(* CODESYS project Checkers.project

Project tree, tasks and I/O mapping:
  Device : PAC320-CXX2X-XX, Parker Hannifin, order no. PAC320-CXX2X-XX, version 3.5.9.10
    application Application
      libraries: Standard, * (System)
      task MainTask (externalevent, external event EVENT_ECM_DC, priority 0) calls EtherCAT_Master.EtherCAT_Task [EtherCAT_Master.EtherCAT_Task], Gameplay, TurnEnforcer, KingTextControl, TestPower, MakeMove, AxisPositionFeedback
      task VISU_TASK (cyclic, interval 100 ms, priority 31) calls VisuElems.Visu_Prg
      data type Piece
      data type BoardSpace
      program HMISequence [SFC]
      visualisation Loading_Screen
      visualisation Home_Screen
      program Gameplay [ST]
      function placePiece [ST]
      program ProgramFlow [SFC]
      visualisation Checkerboard
      function movePieceToStart [ST]
      program Init [ST]
      function pop [ST]
      function assignStartingPositions [ST]
      function checkForJumpRed1 [ST]
      function movePiece [ST]
      function pieceSelect [ST]
      function checkForJumpRed2 [ST]
      global variables GVL
      program TurnEnforcer [ST]
      program MakeMove [ST]
      program UpdateValidMoveArrays [ST]
      function checkForJumpRed3 [ST]
      function checkForJumpRed4 [ST]
      program ClearTakenPieces [ST]
      function checkForJumpBlack1 [ST]
      function checkForJumpBlack2 [ST]
      function checkForJumpBlack3 [ST]
      function checkForJumpBlack4 [ST]
      data type JumpProfile
      function clearJumpArr [ST]
      program KingTextControl [ST]
      program JumpPieces [ST]
      data type JumpDetail
      function push [ST]
      function clearGlobalStack [ST]
      function findSelectedPiece [ST]
      program MakeJump [ST]
      function findPieceAtGivenLocation [ST]
      function clearPieceJumpArray [ST]
      axis group XYZ: TRAFO.Kin_Gantry3, axes X, Y, Z
      SymbolConfiguration
      function block MovePieceMotion [CFC]
      program TestPower [CFC]
      program AxisPositionFeedback [CFC]
      function block timeDelay [CFC]
    SoftMotion General Axis Pool
    EtherCAT_Master : PAC320 EtherCAT Master, Parker Hannifin, order no. PAC320-XXXXX-XX, version 3.5.9.10
      PAC320_BusCoupler : PAC320 BusCoupler, Parker Hannifin, version Revision=16#00000001
          settings: StationAlias = 0; DC sync0 cycletime = 4000; DC sync1 cycletime = 4000
        PACIO_DI16_DO16 : DI16/DO16 1ms 0.5A (PACIO-450-03), Parker Hannifin, version Revision=16#00000001
            settings: StationAlias = 0; DC sync0 cycletime = 4000; DC sync1 cycletime = 4000
            unmapped channels: DigitalOutput0, DigitalOutput1, DigitalOutput2, DigitalOutput3, DigitalOutput4, DigitalOutput5, DigitalOutput6, DigitalOutput7, DigitalOutput8, DigitalOutput9, DigitalOutput10, DigitalOutput11, DigitalOutput12, DigitalOutput13, DigitalOutput14, DigitalOutput15, DigitalInput0, DigitalInput1, DigitalInput2, DigitalInput3, DigitalInput4, DigitalInput5, DigitalInput6, DigitalInput7, DigitalInput8, DigitalInput9, DigitalInput10, DigitalInput11, DigitalInput12, DigitalInput13, DigitalInput14, DigitalInput15
        PACIO_DI16_DO16_1 : DI16/DO16 1ms 0.5A LS (PACIO-450-13), Parker Hannifin, version Revision=16#00000001
            settings: DC sync0 cycletime = 4000; DC sync1 cycletime = 4000
            output GripperMove : BIT  // DigitalOutput0
            unmapped channels: DigitalOutput1, DigitalOutput2, DigitalOutput3, DigitalOutput4, DigitalOutput5, DigitalOutput6, DigitalOutput7, DigitalOutput8, DigitalOutput9, DigitalOutput10, DigitalOutput11, DigitalOutput12, DigitalOutput13, DigitalOutput14, DigitalOutput15, DigitalInput0, DigitalInput1, DigitalInput2, DigitalInput3, DigitalInput4, DigitalInput5, DigitalInput6, DigitalInput7, DigitalInput8, DigitalInput9, DigitalInput10, DigitalInput11, DigitalInput12, DigitalInput13, DigitalInput14, DigitalInput15
      PD_xxC_Standard_EtherCAT_drive : PD-xxC - Standard EtherCAT drive(CoE,EoE,FoE) V2.0, Parker Hannifin, version Revision=16#00000002
          settings: StationAlias = 0; DC sync0 cycletime = 4000
          unmapped channels: Controlword, Target Position, Touch Probe Function, Digital Ouputs, Statusword, Position Actual Value, Following Error Actual Value, Touch Probe Status, Touch Probe 1 Positive Edge Position Value, Digital Inputs
        X : SM_Drive_GenericDSP402, 3S - Smart Software Solutions GmbH, order no. 0, version 4.0.0.0
            settings: wDriveID = 0; dwRatioTechUnitsDenom = 3670016; iRatioTechUnitsNum = -125; fSWMaxVelocity = 100; ScalingIncs = 524288; ScalingMotorTurns2 = 7; ScalingUnits = 125; InvertDirection = TRUE; AdrOffset_8010 = 4; BitOffset_8010 = 0; BitLength_8010 = 16; Address_8010 = '%QW2'; Type_8010 = 'UINT'; AddressPointer_8010 = ADR(%QW2); AdrOffset_8020 = 8; BitOffset_8020 = 0; BitLength_8020 = 32; Address_8020 = '%QD2'; Type_8020 = 'DINT'; AddressPointer_8020 = ADR(%QD2); AdrOffset_8030 = 4294967295; BitOffset_8030 = 0; BitLength_8030 = 0; Address_8030 = ''; Type_8030 = ''; AddressPointer_8030 = 0; AdrOffset_8040 = 4294967295; BitOffset_8040 = 0; BitLength_8040 = 0; Address_8040 = ''; Type_8040 = ''; AddressPointer_8040 = 0; AdrOffset_8050 = 4294967295; BitOffset_8050 = 0; BitLength_8050 = 0; Address_8050 = ''; Type_8050 = ''; AddressPointer_8050 = 0; AdrOffset_8060 = 12; BitOffset_8060 = 0;
              BitLength_8060 = 16; Address_8060 = '%QW6'; Type_8060 = 'UINT'; AddressPointer_8060 = ADR(%QW6); AdrOffset_8070 = 4294967295; BitOffset_8070 = 0; BitLength_8070 = 0; Address_8070 = ''; Type_8070 = ''; AddressPointer_8070 = 0; AdrOffset_8080 = 4294967295; BitOffset_8080 = 0; BitLength_8080 = 0; Address_8080 = ''; Type_8080 = ''; AddressPointer_8080 = 0; AdrOffset_8090 = 16; BitOffset_8090 = 0; BitLength_8090 = 32; Address_8090 = '%QD4'; Type_8090 = 'UDINT'; AddressPointer_8090 = ADR(%QD4); AdrOffset_8510 = 4; BitOffset_8510 = 0; BitLength_8510 = 16; Address_8510 = '%IW2'; Type_8510 = 'UINT'; AddressPointer_8510 = ADR(%IW2); AdrOffset_8520 = 8; BitOffset_8520 = 0; BitLength_8520 = 32; Address_8520 = '%ID2'; Type_8520 = 'DINT'; AddressPointer_8520 = ADR(%ID2); AdrOffset_8530 = 4294967295; BitOffset_8530 = 0; BitLength_8530 = 0; Address_8530 = ''; Type_8530 = ''; AddressPointer_8530 = 0;
              AdrOffset_8540 = 4294967295; BitOffset_8540 = 0; BitLength_8540 = 0; Address_8540 = ''; Type_8540 = ''; AddressPointer_8540 = 0; AdrOffset_8550 = 4294967295; BitOffset_8550 = 0; BitLength_8550 = 0; Address_8550 = ''; Type_8550 = ''; AddressPointer_8550 = 0; AdrOffset_8560 = 24; BitOffset_8560 = 0; BitLength_8560 = 32; Address_8560 = '%ID6'; Type_8560 = 'UDINT'; AddressPointer_8560 = ADR(%ID6); AdrOffset_8570 = 16; BitOffset_8570 = 0; BitLength_8570 = 16; Address_8570 = '%IW8'; Type_8570 = 'UINT'; AddressPointer_8570 = ADR(%IW8); AdrOffset_8580 = 20; BitOffset_8580 = 0; BitLength_8580 = 32; Address_8580 = '%ID5'; Type_8580 = 'DINT'; AddressPointer_8580 = ADR(%ID5); AdrOffset_8590 = 4294967295; BitOffset_8590 = 0; BitLength_8590 = 0; Address_8590 = ''; Type_8590 = ''; AddressPointer_8590 = 0; AdrOffset_8600 = 4294967295; BitOffset_8600 = 0; BitLength_8600 = 0; Address_8600 = '';
              Type_8600 = ''; AddressPointer_8600 = 0; AdrOffset_8600 = 4294967295; BitOffset_8600 = 0; BitLength_8600 = 0; Address_8610 = ''; Type_8610 = ''; AddressPointer_8610 = 0; AdrOffset_8620 = 12; BitOffset_8620 = 0; BitLength_8620 = 32; Address_8620 = '%ID3'; Type_8620 = 'DINT'; AddressPointer_8620 = ADR(%ID3)
      PD_xxC_Standard_EtherCAT_drive_1 : PD-xxC - Standard EtherCAT drive(CoE,EoE,FoE) V2.0, Parker Hannifin, version Revision=16#00000002
          settings: StationAlias = 0; DC sync0 cycletime = 4000
          unmapped channels: Controlword, Target Position, Touch Probe Function, Digital Ouputs, Statusword, Position Actual Value, Following Error Actual Value, Touch Probe Status, Touch Probe 1 Positive Edge Position Value, Digital Inputs
        Y : SM_Drive_GenericDSP402, 3S - Smart Software Solutions GmbH, order no. 0, version 4.0.0.0
            settings: dwRatioTechUnitsDenom = 65536; iRatioTechUnitsNum = 3; fSWMaxVelocity = 100; ScalingIncs = 262144; ScalingMotorTurns2 = 5; ScalingUnits = 60; AdrOffset_8010 = 20; BitOffset_8010 = 0; BitLength_8010 = 16; Address_8010 = '%QW10'; Type_8010 = 'UINT'; AddressPointer_8010 = ADR(%QW10); AdrOffset_8020 = 24; BitOffset_8020 = 0; BitLength_8020 = 32; Address_8020 = '%QD6'; Type_8020 = 'DINT'; AddressPointer_8020 = ADR(%QD6); AdrOffset_8030 = 4294967295; BitOffset_8030 = 0; BitLength_8030 = 0; Address_8030 = ''; Type_8030 = ''; AddressPointer_8030 = 0; AdrOffset_8040 = 4294967295; BitOffset_8040 = 0; BitLength_8040 = 0; Address_8040 = ''; Type_8040 = ''; AddressPointer_8040 = 0; AdrOffset_8050 = 4294967295; BitOffset_8050 = 0; BitLength_8050 = 0; Address_8050 = ''; Type_8050 = ''; AddressPointer_8050 = 0; AdrOffset_8060 = 28; BitOffset_8060 = 0; BitLength_8060 = 16; Address_8060 = '%QW14';
              Type_8060 = 'UINT'; AddressPointer_8060 = ADR(%QW14); AdrOffset_8070 = 4294967295; BitOffset_8070 = 0; BitLength_8070 = 0; Address_8070 = ''; Type_8070 = ''; AddressPointer_8070 = 0; AdrOffset_8080 = 4294967295; BitOffset_8080 = 0; BitLength_8080 = 0; Address_8080 = ''; Type_8080 = ''; AddressPointer_8080 = 0; AdrOffset_8090 = 32; BitOffset_8090 = 0; BitLength_8090 = 32; Address_8090 = '%QD8'; Type_8090 = 'UDINT'; AddressPointer_8090 = ADR(%QD8); AdrOffset_8510 = 28; BitOffset_8510 = 0; BitLength_8510 = 16; Address_8510 = '%IW14'; Type_8510 = 'UINT'; AddressPointer_8510 = ADR(%IW14); AdrOffset_8520 = 32; BitOffset_8520 = 0; BitLength_8520 = 32; Address_8520 = '%ID8'; Type_8520 = 'DINT'; AddressPointer_8520 = ADR(%ID8); AdrOffset_8530 = 4294967295; BitOffset_8530 = 0; BitLength_8530 = 0; Address_8530 = ''; Type_8530 = ''; AddressPointer_8530 = 0; AdrOffset_8540 = 4294967295; BitOffset_8540 = 0;
              BitLength_8540 = 0; Address_8540 = ''; Type_8540 = ''; AddressPointer_8540 = 0; AdrOffset_8550 = 4294967295; BitOffset_8550 = 0; BitLength_8550 = 0; Address_8550 = ''; Type_8550 = ''; AddressPointer_8550 = 0; AdrOffset_8560 = 48; BitOffset_8560 = 0; BitLength_8560 = 32; Address_8560 = '%ID12'; Type_8560 = 'UDINT'; AddressPointer_8560 = ADR(%ID12); AdrOffset_8570 = 40; BitOffset_8570 = 0; BitLength_8570 = 16; Address_8570 = '%IW20'; Type_8570 = 'UINT'; AddressPointer_8570 = ADR(%IW20); AdrOffset_8580 = 44; BitOffset_8580 = 0; BitLength_8580 = 32; Address_8580 = '%ID11'; Type_8580 = 'DINT'; AddressPointer_8580 = ADR(%ID11); AdrOffset_8590 = 4294967295; BitOffset_8590 = 0; BitLength_8590 = 0; Address_8590 = ''; Type_8590 = ''; AddressPointer_8590 = 0; AdrOffset_8600 = 4294967295; BitOffset_8600 = 0; BitLength_8600 = 0; Address_8600 = ''; Type_8600 = ''; AddressPointer_8600 = 0;
              AdrOffset_8600 = 4294967295; BitOffset_8600 = 0; BitLength_8600 = 0; Address_8610 = ''; Type_8610 = ''; AddressPointer_8610 = 0; AdrOffset_8620 = 36; BitOffset_8620 = 0; BitLength_8620 = 32; Address_8620 = '%ID9'; Type_8620 = 'DINT'; AddressPointer_8620 = ADR(%ID9)
      PD_xxC_Standard_EtherCAT_drive_2 : PD-xxC - Standard EtherCAT drive(CoE,EoE,FoE) V2.0, Parker Hannifin, version Revision=16#00000002
          settings: StationAlias = 0; DC sync0 cycletime = 4000
          unmapped channels: Controlword, Target Position, Touch Probe Function, Digital Ouputs, Statusword, Position Actual Value, Following Error Actual Value, Touch Probe Status, Touch Probe 1 Positive Edge Position Value, Digital Inputs
        Z : SM_Drive_GenericDSP402, 3S - Smart Software Solutions GmbH, order no. 0, version 4.0.0.0
            settings: wDriveID = 2; dwRatioTechUnitsDenom = 262144; iRatioTechUnitsNum = 5; fSWMaxVelocity = 100; fSWMaxAcceleration = 500; fSWMaxDeceleration = 500; fSWMaxJerk = 5000; ScalingIncs = 262144; ScalingUnits = 5; AdrOffset_8010 = 36; BitOffset_8010 = 0; BitLength_8010 = 16; Address_8010 = '%QW18'; Type_8010 = 'UINT'; AddressPointer_8010 = ADR(%QW18); AdrOffset_8020 = 40; BitOffset_8020 = 0; BitLength_8020 = 32; Address_8020 = '%QD10'; Type_8020 = 'DINT'; AddressPointer_8020 = ADR(%QD10); AdrOffset_8030 = 4294967295; BitOffset_8030 = 0; BitLength_8030 = 0; Address_8030 = ''; Type_8030 = ''; AddressPointer_8030 = 0; AdrOffset_8040 = 4294967295; BitOffset_8040 = 0; BitLength_8040 = 0; Address_8040 = ''; Type_8040 = ''; AddressPointer_8040 = 0; AdrOffset_8050 = 4294967295; BitOffset_8050 = 0; BitLength_8050 = 0; Address_8050 = ''; Type_8050 = ''; AddressPointer_8050 = 0; AdrOffset_8060 = 44;
              BitOffset_8060 = 0; BitLength_8060 = 16; Address_8060 = '%QW22'; Type_8060 = 'UINT'; AddressPointer_8060 = ADR(%QW22); AdrOffset_8070 = 4294967295; BitOffset_8070 = 0; BitLength_8070 = 0; Address_8070 = ''; Type_8070 = ''; AddressPointer_8070 = 0; AdrOffset_8080 = 4294967295; BitOffset_8080 = 0; BitLength_8080 = 0; Address_8080 = ''; Type_8080 = ''; AddressPointer_8080 = 0; AdrOffset_8090 = 48; BitOffset_8090 = 0; BitLength_8090 = 32; Address_8090 = '%QD12'; Type_8090 = 'UDINT'; AddressPointer_8090 = ADR(%QD12); AdrOffset_8510 = 52; BitOffset_8510 = 0; BitLength_8510 = 16; Address_8510 = '%IW26'; Type_8510 = 'UINT'; AddressPointer_8510 = ADR(%IW26); AdrOffset_8520 = 56; BitOffset_8520 = 0; BitLength_8520 = 32; Address_8520 = '%ID14'; Type_8520 = 'DINT'; AddressPointer_8520 = ADR(%ID14); AdrOffset_8530 = 4294967295; BitOffset_8530 = 0; BitLength_8530 = 0; Address_8530 = ''; Type_8530 = '';
              AddressPointer_8530 = 0; AdrOffset_8540 = 4294967295; BitOffset_8540 = 0; BitLength_8540 = 0; Address_8540 = ''; Type_8540 = ''; AddressPointer_8540 = 0; AdrOffset_8550 = 4294967295; BitOffset_8550 = 0; BitLength_8550 = 0; Address_8550 = ''; Type_8550 = ''; AddressPointer_8550 = 0; AdrOffset_8560 = 72; BitOffset_8560 = 0; BitLength_8560 = 32; Address_8560 = '%ID18'; Type_8560 = 'UDINT'; AddressPointer_8560 = ADR(%ID18); AdrOffset_8570 = 64; BitOffset_8570 = 0; BitLength_8570 = 16; Address_8570 = '%IW32'; Type_8570 = 'UINT'; AddressPointer_8570 = ADR(%IW32); AdrOffset_8580 = 68; BitOffset_8580 = 0; BitLength_8580 = 32; Address_8580 = '%ID17'; Type_8580 = 'DINT'; AddressPointer_8580 = ADR(%ID17); AdrOffset_8590 = 4294967295; BitOffset_8590 = 0; BitLength_8590 = 0; Address_8590 = ''; Type_8590 = ''; AddressPointer_8590 = 0; AdrOffset_8600 = 4294967295; BitOffset_8600 = 0; BitLength_8600 = 0;
              Address_8600 = ''; Type_8600 = ''; AddressPointer_8600 = 0; AdrOffset_8600 = 4294967295; BitOffset_8600 = 0; BitLength_8600 = 0; Address_8610 = ''; Type_8610 = ''; AddressPointer_8610 = 0; AdrOffset_8620 = 60; BitOffset_8620 = 0; BitLength_8620 = 32; Address_8620 = '%ID15'; Type_8620 = 'DINT'; AddressPointer_8620 = ADR(%ID15)
  text list GlobalTextList
*)

// Device/Application/Piece
TYPE Piece :
STRUCT
	isBlack : BOOL := FALSE; // False indicates that a piece is red; true indicates black
	isTaken : BOOL := FALSE; // False indicates that a piece is still in play
	isKing : BOOL := FALSE; // True indicates that a piece is a king
	isSelected : BOOL := FALSE;
	oldLocation : ARRAY [0..1] OF INT := [0,0];
	currentLocation : ARRAY [0..1] OF INT := [0,0]; // -1, -1 indicated that the piece has been taken
	translatedLocation : ARRAY [0..1] OF INT; // translated movement in terms of HMI coordinates
	startingLocation : ARRAY [0..1] OF INT;
	validMoveArr : ARRAY [0..7,0..7] OF BOOL; // 2D array represents the board, true indicates that a piece can move to that space 
	
	jumpArr : ARRAY [0..20,0..3] OF JumpDetail;
	
	startStack : INT;
	jumpedPieceIndex : INT;
	kingText : WSTRING := "";
END_STRUCT
END_TYPE

// Device/Application/BoardSpace
TYPE BoardSpace :
STRUCT
	isBlack : BOOL := FALSE;
	isRed : BOOL := FALSE;
	isEmpty : BOOL := TRUE;
	chosenForMove : BOOL := FALSE;
	
	xLoc : INT;
END_STRUCT
END_TYPE

// Device/Application/JumpProfile
TYPE JumpProfile :
STRUCT
	jumpRef : INT;
	lastJumpRef : INT := -1;
	xMoveLocation : INT;
	yMoveLocation : INT;
	xJumpedLocation : INT;
	yJumpedLocation : INT;
	numPiecesToJump : INT;
	jumpedPieceColor : INT;
	jumpedPieceIndex : INT;
	jumpingPieceX : INT;
	jumpingPieceY : INT;
END_STRUCT
END_TYPE

// Device/Application/JumpDetail
TYPE JumpDetail :
STRUCT
	
	xMoveLocation : INT := -1;
	yMoveLocation : INT := -1;
	jumpedColor : INT := -1;
	jumpedIndex : INT := -1;
	
	
END_STRUCT
END_TYPE

// Device/Application/GVL
{attribute 'qualified_only'}
VAR_GLOBAL
	selectedPieceValidMoveArr : ARRAY [0..7,0..7] OF BOOL;
	noValidMoveArr : ARRAY [0..7,0..7] OF BOOL;
	selectedPieceValidJumpArr : ARRAY [0..7,0..7] OF BOOL;
	board : ARRAY [0..7,0..7] OF BoardSpace; // represents every space on the board
	pieces : ARRAY [0..1,0..11] OF Piece; // 1,x is any black piece, 0,x is any red piece
	redsTurn : BOOL := TRUE;
	
	jumpMoveArr : ARRAY[0..100] OF JumpProfile;
	currentJumpRef : INT := 0;
	
	xMoveSpace : INT := -1;
	yMoveSpace : INT := -1;
	
	boardIsSetup : BOOL;
	
	takenList : ARRAY [0..20,0..1] OF INT;
	takenListLength : INT;
	emptyTakenList : ARRAY [0..20,0..1] OF INT;
	
	jumpStack : ARRAY[0..3] OF JumpDetail;
	currentStackIndex : INT;
	currentJumpProfileNum : INT;
	
	emptyJumpArr : ARRAY [0..20,0..3] OF JumpDetail;
	
	redStack0Offset : ARRAY [0..1] OF INT := [0,100]; // coordinate offset of red stacks in HMI (at beginning of game)
	redStack1Offset : ARRAY [0..1] OF INT := [100,100]; // coordinate offset of red stacks in HMI (at beginning of game)
	redStack2Offset : ARRAY [0..1] OF INT := [200, 100]; // coordinate offset of red stacks in HMI (at beginning of game)
	
	blackStack0Offset : ARRAY [0..1] OF INT := [350,-450];
	blackStack1Offset : ARRAY [0..1] OF INT := [250,-450];
	blackStack2Offset : ARRAY [0..1] OF INT := [150,-450];
	
	redPiecesTaken : INT := 0;
	blackPiecesTaken : INT := 0;
	
	test : BOOL := FALSE;
	
END_VAR

// Device/Application/Gameplay
PROGRAM Gameplay
VAR
	//selectedPieceValidMoveArr : ARRAY [0..7,0..7] OF BOOL;
	//noValidMoveArr : ARRAY [0..7,0..7] OF BOOL;
	//board : ARRAY [0..7,0..7] OF BoardSpace; // represents every space on the board
	//pieces : ARRAY [0..1,0..11] OF Piece; // 0,x is any black piece, 1,x is any red piece
	startingPositionsRed : ARRAY [0..1,0..11] OF INT;
	startingPositionsBlack : ARRAY [0..1,0..11] OF INT;
	redIsAssigned : BOOL := FALSE;
	blackIsAssigned : BOOL := FALSE;
	
	// ****************VARIABLES FOR BOARD SETUP*******************
	numStacks : INT := 3;
	numPiecesInStack : INT := 5;
	numPieces : INT := 12;
	currentStack : INT := 0; // stack that gripper is currently drawing from
	currentPiece : INT := 0; // piece number that gripper has set up
	currentStackPos : INT := 0;	// stack position flows 0-4 from top to bottom
	currentSpace : ARRAY [0..1] OF INT;
	piecePosition : ARRAY[0..1] OF INT;
	
	done : BOOL;
	i : INT := 0;
	j : INT := 0;
	boardCleared : BOOL := FALSE;
	y: INT;
	pieceNum: INT;
	x: INT;
	temp : INT;
	commenceSetup : BOOL := FALSE; // Variable toggled by pushing the set up board button
	xPos: INT;
	yPos: INT;
	found : BOOL := FALSE;
END_VAR

IF(commenceSetup) THEN
	IF(NOT GVL.boardIsSetup) THEN
	

		// Assigns starting positions for red and black GVL.pieces
	IF(NOT redIsAssigned) THEN
		startingPositionsRed := assignStartingPositions(startingPositionsRed, TRUE);
		redIsAssigned := TRUE;
	END_IF
	IF(NOT blackIsAssigned) THEN
		startingPositionsBlack := assignStartingPositions(startingPositionsBlack, FALSE);
		blackIsAssigned := TRUE;
	END_IF


	// initializes values for red GVL.pieces
	FOR i := 0 TO (numPieces - 1) DO
		GVL.pieces[0,i].isBlack := FALSE;
		GVL.pieces[0,i].isKing := FALSE;
		GVL.pieces[0,i].isTaken := FALSE;
		GVL.pieces[0,i].currentLocation[0] := startingPositionsRed[0,i]; 
		GVL.pieces[0,i].currentLocation[1] := startingPositionsRed[1,i];
		GVL.pieces[0,i].jumpedPieceIndex := i;
		IF(i < numPiecesInStack) THEN
			GVL.pieces[0,i].startStack := 0;
		ELSIF(i < (numPiecesInStack * 2) AND i >= numPiecesInStack) THEN
			GVL.pieces[0,i].startStack := 1;
		ELSE
			GVL.pieces[0,i].startStack := 2;
		END_IF
		GVL.pieces[0,i] := movePieceToStart(GVL.pieces[0,i]);
		GVL.board[GVL.pieces[0,i].currentLocation[0], GVL.pieces[0,i].currentLocation[1]].isRed := TRUE;
		GVL.board[GVL.pieces[0,i].currentLocation[0], GVL.pieces[0,i].currentLocation[1]].isBlack := FALSE;
		GVL.board[GVL.pieces[0,i].currentLocation[0], GVL.pieces[0,i].currentLocation[1]].isEmpty := FALSE;
	END_FOR


	// initializes values for black GVL.pieces
	FOR i := 0 TO (numPieces - 1) DO
		GVL.pieces[1,i].isBlack := TRUE;
		GVL.pieces[1,i].isKing := FALSE;
		GVL.pieces[1,i].isTaken := FALSE;
		GVL.pieces[1,i].currentLocation[0] := startingPositionsBlack[0,i];
		GVL.pieces[1,i].currentLocation[1] := startingPositionsBlack[1,i];
		IF(i < numPiecesInStack) THEN
			GVL.pieces[1,i].startStack := 0;
		ELSIF(i < (numPiecesInStack * 2) AND i >= numPiecesInStack) THEN
			GVL.pieces[1,i].startStack := 1;
		ELSE
			GVL.pieces[1,i].startStack := 2;
		END_IF
		GVL.pieces[1,i] := movePieceToStart(GVL.pieces[1,i]);
		GVL.board[GVL.pieces[1,i].currentLocation[0], GVL.pieces[1,i].currentLocation[1]].isRed := FALSE;
		GVL.board[GVL.pieces[1,i].currentLocation[0], GVL.pieces[1,i].currentLocation[1]].isBlack := TRUE;
		GVL.board[GVL.pieces[1,i].currentLocation[0], GVL.pieces[1,i].currentLocation[1]].isEmpty := FALSE;
	END_FOR

	GVL.boardIsSetup := TRUE;
END_IF

// Setup valid moves for red
FOR i:= 0 TO numPieces - 1 DO
	x:= GVL.pieces[0,i].currentLocation[0];
	y := GVL.pieces[0,i].currentLocation[1];
	
	// Checks for move up and right
	IF(x+1 < 8 AND y+1 < 8 AND GVL.board[x+1,y+1].isEmpty) THEN
		GVL.pieces[0,i].validMoveArr[x+1,y+1] := TRUE;
	END_IF

	// Checks for move up and left
	IF(x-1 >= 0 AND y+1 < 8 AND GVL.board[x-1,y+1].isEmpty) THEN
		GVL.pieces[0,i].validMoveArr[x-1,y+1] := TRUE;
	END_IF
	
	IF(x+1 < 8 AND y+1 < 8 AND NOT GVL.board[x+1,y+1].isEmpty AND GVL.board[x+1,y+1].isBlack) THEN
		
		//possible jump
	END_IF
	
END_FOR

// Setup valid moves for black
FOR i:= 0 TO numPieces - 1 DO
	x:= GVL.pieces[1,i].currentLocation[0];
	y := GVL.pieces[1,i].currentLocation[1];
	
	// Checks for move up and right
	IF(x+1 < 8 AND y+1 < 8 AND GVL.board[x+1,y-1].isEmpty) THEN
		GVL.pieces[1,i].validMoveArr[x+1,y-1] := TRUE;
	END_IF

	// Checks for move up and left
	IF(x-1 >= 0 AND y+1 < 8 AND GVL.board[x-1,y-1].isEmpty) THEN
		GVL.pieces[1,i].validMoveArr[x-1,y-1] := TRUE;
	END_IF
	
	(*
	IF(x+1 < 8 AND y+1 < 8 AND NOT GVL.board[x+1,y+1].isEmpty AND GVL.board[x+1,y+1].isBlack) THEN
		
		//possible jump
	END_IF
	*)
	
END_FOR



END_IF

END_PROGRAM

// Device/Application/assignStartingPositions
FUNCTION assignStartingPositions : ARRAY [0..1,0..11] OF INT;
VAR_INPUT
	startingPos : ARRAY [0..1,0..11] OF INT;
	isRed : BOOL;
END_VAR
VAR
	numPieces : INT := 12;
	
	i: INT;
	y: INT;
	x: INT;
	temp: INT;
END_VAR

IF(isRed) THEN
	FOR i := 0 TO (numPieces - 1) DO 	
		y := i / 4;
		x := ((2 * i) MOD 8) + (y MOD 2);
		startingPos[0,i] := x;
		startingPos[1,i] := y;
	END_FOR
ELSE
	FOR i := 0 TO (numPieces - 1) DO 
		temp := i / 4;
		x := ((2 * i) MOD 8) + (temp MOD 2);
		y := temp + 5;
		x := x + 1;
		IF(x >= 8) THEN
			x := x MOD 8;
		END_IF
		startingPos[0,i] := x;
		startingPos[1,i] := y;	
	END_FOR
END_IF

assignStartingPositions := startingPos;
RETURN;

END_FUNCTION

// Device/Application/movePieceToStart
FUNCTION movePieceToStart : Piece
VAR_INPUT
	currentPiece : Piece;
END_VAR
VAR
	
	spaceTranslation : ARRAY [0..1] OF INT; // small numbers (0-7) that indicate how many spaces a piece needs to be moved
	sizeOfMoveX : INT := 50;
	sizeOfMoveY : INT := -50;
END_VAR

movePieceToStart := currentPiece;
IF(NOT movePieceToStart.isBlack) THEN
	// Moves pieces from their stack to the origin (board sqaure 0,0 or bottom left corner)
	IF(currentPiece.startStack = 0) THEN
		movePieceToStart.translatedLocation[0] := currentPiece.translatedLocation[0] - GVL.redStack0Offset[0];
		movePieceToStart.translatedLocation[1] := currentPiece.translatedLocation[1] - GVL.redStack0Offset[1];
		
	ELSIF(currentPiece.startStack = 1) THEN
		movePieceToStart.translatedLocation[0] := currentPiece.translatedLocation[0] - GVL.redStack1Offset[0];
		movePieceToStart.translatedLocation[1] := currentPiece.translatedLocation[1] - GVL.redStack1Offset[1];
	ELSE
		movePieceToStart.translatedLocation[0] := currentPiece.translatedLocation[0] - GVL.redStack2Offset[0];
		movePieceToStart.translatedLocation[1] := currentPiece.translatedLocation[1] - GVL.redStack2Offset[1];
	END_IF
ELSE
	IF(currentPiece.startStack = 0) THEN
		movePieceToStart.translatedLocation[0] := currentPiece.translatedLocation[0] - GVL.blackStack0Offset[0];
		movePieceToStart.translatedLocation[1] := currentPiece.translatedLocation[1] - GVL.blackStack0Offset[1];
	ELSIF(currentPiece.startStack = 1) THEN
		movePieceToStart.translatedLocation[0] := currentPiece.translatedLocation[0] - GVL.blackStack1Offset[0];
		movePieceToStart.translatedLocation[1] := currentPiece.translatedLocation[1] - GVL.blackStack1Offset[1];
	ELSE
		movePieceToStart.translatedLocation[0] := currentPiece.translatedLocation[0] - GVL.blackStack2Offset[0];
		movePieceToStart.translatedLocation[1] := currentPiece.translatedLocation[1] - GVL.blackStack2Offset[1];
	END_IF			

END_IF

movePieceToStart.startingLocation := movePieceToStart.translatedLocation;

spaceTranslation[0] := movePieceToStart.currentLocation[0] - movePieceToStart.oldLocation[0];
spaceTranslation[1] := movePieceToStart.currentLocation[1] - movePieceToStart.oldLocation[1];

movePieceToStart.translatedLocation[0] := movePieceToStart.translatedLocation[0] + (spaceTranslation[0] * sizeOfMoveX);
movePieceToStart.translatedLocation[1] := movePieceToStart.translatedLocation[1] + (spaceTranslation[1] * sizeOfMoveY);

// set oldLocation to currentLocation
movePieceToStart.oldLocation[0] := movePieceToStart.currentLocation[0];
movePieceToStart.oldLocation[1] := movePieceToStart.currentLocation[1];


RETURN;

END_FUNCTION

// Device/Application/TurnEnforcer
PROGRAM TurnEnforcer
VAR
	i : INT;
	wrongColorSelected : BOOL;
END_VAR

// Stops user from selecting a piece that is taken
FOR i := 0 TO 11 DO
	IF(GVL.pieces[1,i].isTaken)THEN 
		GVL.pieces[1,i].isSelected := FALSE;
	ELSIF(GVL.pieces[0,i].isTaken) THEN
		GVL.pieces[0,i].isSelected := FALSE;
	END_IF
END_FOR

// Stops user from picking the wrong color
wrongColorSelected := FALSE;

IF(GVL.redsTurn) THEN
	FOR i := 0 TO 11 DO
		IF(GVL.pieces[1,i].isSelected)THEN 
			 GVL.pieces[1,i].isSelected := FALSE;
			 wrongColorSelected := TRUE;
		END_IF
	END_FOR
ELSE
	FOR i := 0 TO 11 DO
		IF(GVL.pieces[0,i].isSelected)THEN 
			 GVL.pieces[0,i].isSelected := FALSE;
			 wrongColorSelected := TRUE;
		END_IF				
	END_FOR
END_IF

IF(wrongColorSelected) THEN
	GVL.selectedPieceValidMoveArr := GVL.noValidMoveArr;
END_IF

END_PROGRAM

// Device/Application/KingTextControl
PROGRAM KingTextControl
VAR
	i : INT;
END_VAR

FOR i := 0 TO 11 DO
	IF(GVL.pieces[0,i].isKing) THEN
		GVL.pieces[0,i].kingText := "K";
	END_IF
	IF(GVL.pieces[1,i].isKing) THEN
		GVL.pieces[1,i].kingText := "K";
	END_IF
END_FOR

END_PROGRAM

// Device/Application/TestPower
PROGRAM TestPower
VAR
	xPower: MC_Power;
	yPower: MC_Power;
	zPower: MC_Power;
	EnableAxes: MC_GroupEnable;
	Enable: BOOL;
END_VAR

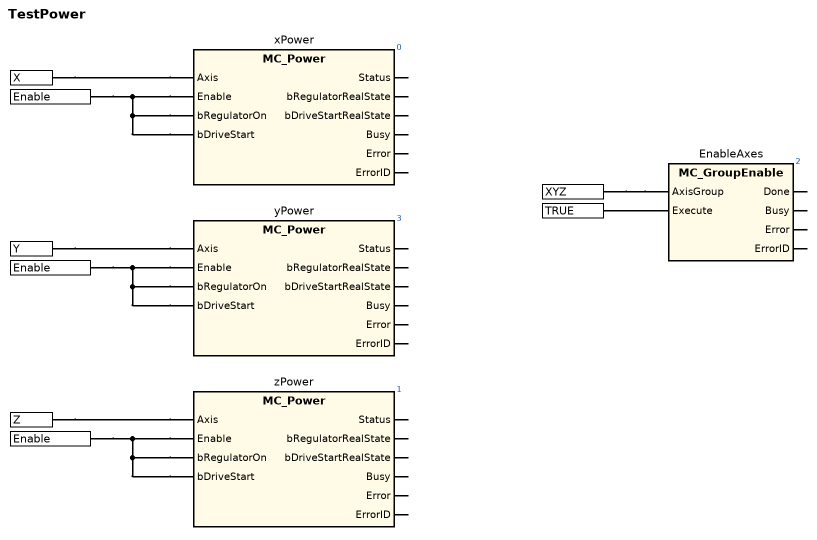
xPower(Axis := X, Enable := Enable, bRegulatorOn := Enable, bDriveStart := Enable); // MC_Power
zPower(Axis := Z, Enable := Enable, bRegulatorOn := Enable, bDriveStart := Enable); // MC_Power
EnableAxes(AxisGroup := XYZ, Execute := TRUE); // MC_GroupEnable
yPower(Axis := Y, Enable := Enable, bRegulatorOn := Enable, bDriveStart := Enable); // MC_Power

END_PROGRAM

// Device/Application/MakeMove
PROGRAM MakeMove
// moveSpace variables are only changed when a square is pushed in the HMI
VAR
	i : INT;
	counter : INT;
	xCurrentSpace : INT;
	yCurrentSpace : INT;
	currentPiece : Piece;
	selected : BOOL;
	redOrBlack : INT;
	jumpedPieceIndex : INT;
	
	spaceTranslation : ARRAY [0..1] OF INT; // small numbers (0-7) that indicate how many spaces a piece needs to be moved
	sizeOfMoveX : INT := 50;
	sizeOfMoveY : INT := -50;
	
	caseState : INT := 000;
	moveTest : MovePieceMotion;
	
	xOffset : LREAL := 100.455;
	yOffset : LREAL := -25.654;
	zUp : LREAL := 15;
	zDown: LREAL := 49;
	
	xStack : LREAL := 111;
	yStack : LREAL := -73;
	pieceOffset : LREAL := 6.36; 
	
	selectedPiece : ARRAY [0..1] OF INT;
	
	xPiece: INT;
	yPiece: INT;
	
	wait : timeDelay;
	
	jumpCounter : INT;

END_VAR

CASE caseState OF

// Will run in this case as long as a move space isn't selected
000:
	IF(GVL.xMoveSpace <> -1 AND GVL.yMoveSpace <> -1) THEN
		//GripperMove := FALSE;
		caseState := 001;
	END_IF
	
// If the move is valid, execution of the move begins by positioning
// the gripper over the piece that is to be moved
// If the move is invalid, case statement jumps back to case 000
001: 
	selectedPiece := findSelectedPiece();
	IF(GVL.selectedPieceValidMoveArr[GVL.xMoveSpace, GVL.yMoveSpace]) THEN
		xPiece := GVL.pieces[selectedPiece[0],selectedPiece[1]].currentLocation[0];
		yPiece := GVL.pieces[selectedPiece[0],selectedPiece[1]].currentLocation[1];
	
		moveTest.xPos := xOffset + (xPiece * 20);
		moveTest.yPos := yOffset + (yPiece * 20);
		moveTest.zPos := zUp;
	
		caseState := 002;
	ELSE
		// Deselects all pieces
		FOR i:=0 TO 11 DO
			GVL.pieces[0,i].isSelected := FALSE;
			GVL.pieces[1,i].isSelected := FALSE;			
		END_FOR
		GVL.xMoveSpace := -1;
		GVL.yMoveSpace := -1;
		
		caseState := 000;
	END_IF

// Move is executed	
002:
	moveTest.ExecuteMove := TRUE;
	caseState := 003;

// Once the gripper is in position above the piece to be moved
// execute move is set to false
003:
	IF(moveTest.MoveDone) THEN
		caseState := 004;
		moveTest.ExecuteMove := FALSE;
	END_IF

// Sets gripper to down position over the current piece
004:
	moveTest.zPos := zDown;
	caseState := 005;

005:
	moveTest.ExecuteMove := TRUE;
	caseState := 006;

// THIS IS WHERE THE PIECE WILL BE PICKED UP	
006:
	IF(moveTest.MoveDone)THEN
		caseState := 007;
		moveTest.ExecuteMove := FALSE;
		GripperMove := TRUE;
		wait.startTimer := TRUE;
	END_IF

007:
	IF(wait.done) THEN
		wait.startTimer := FALSE;
		moveTest.zPos := zUp;
		caseState := 008;
	END_IF
	
008: 
	moveTest.ExecuteMove := TRUE;
	caseState := 009;

009:
	IF(moveTest.MoveDone)THEN
		caseState := 010;
		moveTest.ExecuteMove := FALSE;
	END_IF
	
	
010:
	IF(GVL.xMoveSpace >= 0 AND GVL.yMoveSpace >= 0) THEN
		selected := FALSE;
		i := 0;
		// Figure out which piece is selected
		WHILE(i < 12 AND NOT selected) DO
		
			IF(GVL.pieces[0,i].isSelected) THEN
				xCurrentSpace := GVL.pieces[0,i].currentLocation[0];
				yCurrentSpace := GVL.pieces[0,i].currentLocation[1];
				currentPiece := GVL.pieces[0,i];
				redOrBlack := 0;
				jumpedPieceIndex := i;
				selected := TRUE;
			END_IF
			IF(GVL.pieces[1,i].isSelected) THEN
				xCurrentSpace := GVL.pieces[1,i].currentLocation[0];
				yCurrentSpace := GVL.pieces[1,i].currentLocation[1];
				currentPiece := GVL.pieces[1,i];
				redOrBlack := 1;
				jumpedPieceIndex := i;
				selected := TRUE;
			END_IF
			i := i + 1;
	
		END_WHILE
	
		// Determine if the move is legal
		IF(GVL.selectedPieceValidMoveArr[GVL.xMoveSpace, GVL.yMoveSpace])THEN 
			// Perform the move
			currentPiece.translatedLocation[0] := currentPiece.startingLocation[0] + (GVL.xMoveSpace * sizeOfMoveX);
			currentPiece.translatedLocation[1] := currentPiece.startingLocation[1] + (GVL.yMoveSpace * sizeOfMoveY);;
		
		
			moveTest.xPos := xOffset + (GVL.xMoveSpace * 20);
			moveTest.yPos := yOffset + (GVL.yMoveSpace * 20);
			moveTest.zPos := zUp;

			caseState := 020;
		
		
			// sets pieces current location as the old location, as it is about to move
			currentPiece.oldLocation[0] := currentPiece.currentLocation[0];
			currentPiece.oldLocation[1] := currentPiece.currentLocation[1];
	
			// updates the current location after the move has been completed
			currentPiece.currentLocation[0] := GVL.xMoveSpace;
			currentPiece.currentLocation[1] := GVL.yMoveSpace;
		
			// Piece is red and has achieved king status
			IF(currentPiece.currentLocation[1] = 7 AND NOT currentPiece.isBlack) THEN
				currentPiece.isKing := TRUE;
			// Piece is black and has achieved king status
			ELSIF(currentPiece.currentLocation[1] = 0 AND currentPiece.isBlack) THEN
				currentPiece.isKing := TRUE;
			END_IF
			
		
			// updates board space player just moved from
			GVL.board[currentPiece.oldLocation[0], currentPiece.oldLocation[1]].isEmpty := TRUE;
			GVL.board[currentPiece.oldLocation[0], currentPiece.oldLocation[1]].isBlack := FALSE;
			GVL.board[currentPiece.oldLocation[0], currentPiece.oldLocation[1]].isRed := FALSE;
		
			// updates board space that the player just moved to
			GVL.board[currentPiece.currentLocation[0], currentPiece.currentLocation[1]].isEmpty := FALSE;
			IF(currentPiece.isBlack)THEN
				GVL.board[currentPiece.currentLocation[0], currentPiece.currentLocation[1]].isBlack := TRUE;
				GVL.board[currentPiece.currentLocation[0], currentPiece.currentLocation[1]].isRed := FALSE;
			ELSE
				GVL.board[currentPiece.currentLocation[0], currentPiece.currentLocation[1]].isBlack := FALSE;
				GVL.board[currentPiece.currentLocation[0], currentPiece.currentLocation[1]].isRed := TRUE;
			END_IF
		
			GVL.pieces[redOrBlack, jumpedPieceIndex] := currentPiece;
		
		
		
			// Make it the other persons turn
			IF(GVL.redsTurn) THEN
				GVL.redsTurn := FALSE;
			ELSE
				GVL.redsTurn := TRUE;	
			END_IF
		
		
			MakeJump();
			UpdateValidMoveArrays();
		
			// Deselects all pieces
			GVL.selectedPieceValidMoveArr := GVL.noValidMoveArr;
			FOR i:=0 TO 11 DO
				GVL.pieces[0,i].isSelected := FALSE;
				GVL.pieces[1,i].isSelected := FALSE;			
			END_FOR
		
			IF(currentPiece.oldLocation[0] + 1 = currentPiece.currentLocation[0] OR
				currentPiece.oldLocation[1] + 1 = currentPiece.currentLocation[1] OR
				currentPiece.oldLocation[0] - 1 = currentPiece.currentLocation[0] OR
				currentPiece.oldLocation[1] - 1 = currentPiece.currentLocation[1]) THEN
				// DO NOTHING
			ELSE
				ClearTakenPieces();
			END_IF
		
		
		ELSE
			// Deselects all pieces
			GVL.selectedPieceValidMoveArr := GVL.noValidMoveArr;
			FOR i:=0 TO 11 DO
				GVL.pieces[0,i].isSelected := FALSE;
				GVL.pieces[1,i].isSelected := FALSE;			
			END_FOR
			
			GVL.xMoveSpace := -1;
			GVL.yMoveSpace := -1;
		
			caseState := 000;
			
		END_IF
		clearJumpArr();
		
		GVL.xMoveSpace := -1;
		GVL.yMoveSpace := -1;

		GVL.currentJumpRef := 0;

		//counter := counter + 1;
		

		

			
	END_IF
	
020:
	moveTest.ExecuteMove := TRUE;
	caseState := 030;
	
030:
	IF(moveTest.MoveDone) THEN
		caseState := 031;
		moveTest.ExecuteMove := FALSE;
		UpdateValidMoveArrays();
	END_IF
	

// Sets gripper to down position over the current piece
031:
	moveTest.zPos := zDown;
	caseState := 032;
	
032:
	moveTest.ExecuteMove := TRUE;
	caseState := 033;

// THIS IS WHERE THE PIECE WILL BE DROPPED OFF	
033:	
	IF(moveTest.MoveDone)THEN
		caseState := 034;
		moveTest.ExecuteMove := FALSE;
		GripperMove := FALSE;
		wait.startTimer := TRUE;
	END_IF
	
// Sets gripper to up position over the current piece
034:
	IF(wait.done)THEN
		wait.startTimer := FALSE;
		moveTest.zPos := zUp;
		caseState := 035;
	END_IF
	
035:
	moveTest.ExecuteMove := TRUE;
	caseState := 036;

036:	
	IF(moveTest.MoveDone)THEN
		caseState := 040;
		moveTest.ExecuteMove := FALSE;
		jumpCounter := 0;	
	END_IF
	
	
// Moves over the top of the piece to be jumped
040:
	IF(jumpCounter < GVL.takenListLength) THEN
		xPiece := GVL.takenList[jumpCounter,0];
		yPiece := GVL.takenList[jumpCounter,1];

		moveTest.xPos := xOffset + (xPiece * 20);
		moveTest.yPos := yOffset + (yPiece * 20);
		moveTest.zPos := zUp;
		caseState := 041;
	ELSE
		caseState := 100;	
	END_IF
	
041:
	moveTest.ExecuteMove := TRUE;
	caseState := 042;
	
042:
	IF(moveTest.MoveDone) THEN
		caseState := 043;
		moveTest.ExecuteMove := FALSE;
	END_IF
	
043:
	moveTest.zPos := zDown;
	caseState := 044;
	
044:
	moveTest.ExecuteMove := TRUE;
	caseState := 046;

// THIS IS WHERE THE JUMPED PIECE IS PICKED UP	
046:
	IF(moveTest.MoveDone)THEN
		caseState := 047;
		moveTest.ExecuteMove := FALSE;
		GripperMove := TRUE;
		wait.startTimer := TRUE;
	END_IF

047:
	IF(wait.done) THEN
		wait.startTimer := FALSE;
		moveTest.zPos := zUp;
		caseState := 048;
	END_IF
	
048: 
	moveTest.ExecuteMove := TRUE;
	caseState := 049;

049:
	IF(moveTest.MoveDone)THEN
		caseState := 050;
		moveTest.ExecuteMove := FALSE;
	END_IF	
// PIECE IS GRABBED AND UP

// Moves to stack where piece is to be dropped off
050:
	moveTest.xPos := xStack;
	moveTest.yPos := yStack;
	moveTest.zPos := zUp + (jumpCounter * pieceOffset);
	jumpCounter := jumpCounter + 1;
	caseState := 051;
	
051:
	moveTest.ExecuteMove := TRUE;
	caseState := 052;
	
052:
	IF(moveTest.MoveDone) THEN
		caseState := 053;
		moveTest.ExecuteMove := FALSE;
	END_IF
	
053:
	moveTest.zPos := zDown;
	caseState := 054;

054:
	moveTest.ExecuteMove := TRUE;
	caseState := 055;

// THIS IS WHERE THE PIECE WILL BE DROPPED OFF	
055:
	IF(moveTest.MoveDone)THEN
		caseState := 056;
		moveTest.ExecuteMove := FALSE;
		GripperMove := FALSE;
		wait.startTimer := TRUE;
	END_IF
	
056:
	IF(wait.done)THEN
		wait.startTimer := FALSE;
		moveTest.zPos := zUp;
		caseState := 057;
	END_IF
	
057:
	moveTest.ExecuteMove := TRUE;
	caseState := 058;

058:
	IF(moveTest.MoveDone) THEN
		caseState := 040;
		moveTest.ExecuteMove := FALSE;
	END_IF


100:
	IF(NOT moveTest.ExecuteMove) THEN
		caseState := 000;
	END_IF
	

END_CASE

moveTest(AxisGroup := XYZ);
wait();

END_PROGRAM

// Device/Application/findSelectedPiece
FUNCTION findSelectedPiece : ARRAY [0..1] OF INT
VAR_INPUT
END_VAR
VAR
	i : INT;
END_VAR

FOR i := 0 TO 11 DO
	IF(GVL.pieces[0,i].isSelected) THEN
		findSelectedPiece[0] := 0;
		findSelectedPiece[1] := i;
	END_IF
	IF(GVL.pieces[1,i].isSelected) THEN
		findSelectedPiece[0] := 1;
		findSelectedPiece[1] := i;
	END_IF
END_FOR

RETURN;

END_FUNCTION

// Device/Application/MakeJump
PROGRAM MakeJump
VAR
	pieceColor : INT;
	pieceIndex : INT;
	
	jumpedColor : INT;
	jumpedIndex : INT;
	
	jumpedLocX : INT := -1;
	jumpedLocY : INT := -1;
	
	temp : ARRAY [0..1] OF INT;
	
	i : INT;
	j : INT := 0;
	
	usedJumpProfile : INT;
	lengthJumpSeq : INT := -1;
END_VAR

// Null out global variables that are used when taking pieces that are jumped
GVL.takenList := GVL.emptyTakenList;
GVL.takenListLength := 0;

// Finds the index of the selected piece that is making a move
temp := findSelectedPiece();
pieceColor := temp[0];
pieceIndex := temp[1];

// Finds longest jump profile that ends at the chosen destination space
FOR i := 20 TO 0 BY -1 DO 
	
	j := 0;
	WHILE(j < 4 AND GVL.pieces[pieceColor, pieceIndex].jumpArr[i,j].xMoveLocation <> -1) DO
		IF(GVL.pieces[pieceColor, pieceIndex].jumpArr[i,j].xMoveLocation = GVL.xMoveSpace AND GVL.pieces[pieceColor, pieceIndex].jumpArr[i,j].yMoveLocation = GVL.yMoveSpace AND j > lengthJumpSeq)THEN
			usedJumpProfile := i;
			lengthJumpSeq := j;
		END_IF
		j := j + 1;
	END_WHILE

END_FOR

GVL.takenListLength := lengthJumpSeq + 1;

FOR i := 0 TO lengthJumpSeq DO
	// assigns easy to read values to piece that is to be jumped
	jumpedColor := GVL.pieces[pieceColor, pieceIndex].jumpArr[usedJumpProfile,i].jumpedColor;
	jumpedIndex := GVL.pieces[pieceColor, pieceIndex].jumpArr[usedJumpProfile,i].jumpedIndex;
	IF(jumpedColor >= 0) THEN
		jumpedLocX := GVL.pieces[jumpedColor, jumpedIndex].currentLocation[0];
		jumpedLocY := GVL.pieces[jumpedColor, jumpedIndex].currentLocation[1];
		
		GVL.takenList[i,0] := jumpedLocX;
		GVL.takenList[i,1] := jumpedLocY;
	
		GVL.pieces[jumpedColor, jumpedIndex].translatedLocation[0] := 0;
		GVL.pieces[jumpedColor, jumpedIndex].translatedLocation[1] := 0;
	
		// Nulls out information for all taken pieces
		GVL.pieces[jumpedColor, jumpedIndex].isTaken := TRUE;
		GVL.pieces[jumpedColor, jumpedIndex].isKing := FALSE;
	
		// Makes location an invalid value
		GVL.pieces[jumpedColor, jumpedIndex].currentLocation[0] := -1;
		GVL.pieces[jumpedColor, jumpedIndex].currentLocation[1] := -1;
	
		// Makes the taken piece have zero valid moves
		GVL.pieces[jumpedColor, jumpedIndex].validMoveArr := GVL.noValidMoveArr;
	
		WHILE(jumpedLocX = 0 AND jumpedLocY = 0) DO
			//
		END_WHILE
	
		// Clears board space that was occupied by the taken piece
		GVL.board[jumpedLocX, jumpedLocY].isEmpty := TRUE;
		GVL.board[jumpedLocX, jumpedLocY].isRed := FALSE;
		GVL.board[jumpedLocX, jumpedLocY].isBlack := FALSE;
	END_IF			
END_FOR

END_PROGRAM

// Device/Application/UpdateValidMoveArrays
PROGRAM UpdateValidMoveArrays
VAR
	i : INT;
	x: INT;
	y : INT;
	xNext : INT;
	yNext : INT;
END_VAR

// Code will run continuously, but will not execute until board is setup
// If code runs before board is setup, there will be an error, so don't do that ok?
IF(GVL.boardIsSetup)THEN	
	// Checks moves for red
	IF(GVL.redsTurn) THEN
	GVL.currentJumpRef := 0;
	FOR i:= 0 TO 11 DO
		GVL.pieces[0,i].validMoveArr := GVL.noValidMoveArr;
		x:= GVL.pieces[0,i].currentLocation[0];
		y := GVL.pieces[0,i].currentLocation[1];
	
		// Checks for move up and right
		IF(x+1 < 8 AND y+1 < 8 AND GVL.board[x+1,y+1].isEmpty) THEN
			GVL.pieces[0,i].validMoveArr[x+1,y+1] := TRUE;
		END_IF

		// Checks for move up and left
		IF(x-1 >= 0 AND y+1 < 8 AND GVL.board[x-1,y+1].isEmpty) THEN
			GVL.pieces[0,i].validMoveArr[x-1,y+1] := TRUE;
		END_IF
		
		// Checks for move down and left (FOR KINGS ONLY)
		IF(x-1 >= 0 AND y-1 >= 0 AND GVL.board[x-1,y-1].isEmpty AND GVL.pieces[0,i].isKing) THEN
			GVL.pieces[0,i].validMoveArr[x-1,y-1] := TRUE;
		END_IF
		
		// Checks for move down and right (FOR KINGS ONLY)
		IF(x+1 >= 0 AND y-1 >= 0 AND GVL.board[x+1,y-1].isEmpty AND GVL.pieces[0,i].isKing) THEN
			GVL.pieces[0,i].validMoveArr[x+1,y-1] := TRUE;
		END_IF
		
		// Checks for all red jumps (pseudo recursive call)
		clearGlobalStack();
		GVL.currentStackIndex := 0;
		GVL.currentJumpProfileNum := 0;
		clearPieceJumpArray(0,i);
		GVL.pieces[0,i] := checkForJumpRed1(GVL.pieces[0,i], i);
		
	END_FOR
	
	ELSE
	GVL.currentJumpRef := 0;
	// Setup valid moves for black
	FOR i:= 0 TO 11 DO
		GVL.pieces[1,i].validMoveArr := GVL.noValidMoveArr;
		x:= GVL.pieces[1,i].currentLocation[0];
		y := GVL.pieces[1,i].currentLocation[1];
	
		// Checks for down and right
		IF(x+1 < 8 AND y-1 >= 0 AND GVL.board[x+1,y-1].isEmpty) THEN
			GVL.pieces[1,i].validMoveArr[x+1,y-1] := TRUE;
		END_IF

		// Checks for move down and left
		IF(x-1 >= 0 AND y-1 >= 0 AND GVL.board[x-1,y-1].isEmpty) THEN
			GVL.pieces[1,i].validMoveArr[x-1,y-1] := TRUE;
		END_IF
		
		// Checks for move up and left (FOR KINGS ONLY)
		IF(x-1 >= 0 AND y+1 >= 0 AND GVL.board[x-1,y+1].isEmpty AND GVL.pieces[1,i].isKing) THEN
			GVL.pieces[0,i].validMoveArr[x-1,y+1] := TRUE;
		END_IF
		
		// Checks for move up and right (FOR KINGS ONLY)
		IF(x+1 >= 0 AND y+1 >= 0 AND GVL.board[x+1,y+1].isEmpty AND GVL.pieces[1,i].isKing) THEN
			GVL.pieces[0,i].validMoveArr[x+1,y+1] := TRUE;
		END_IF
	
		clearGlobalStack();
		GVL.currentStackIndex := 0;
		GVL.currentJumpProfileNum := 0;
		clearPieceJumpArray(0,i);
		GVL.pieces[1,i] := checkForJumpBlack1(GVL.pieces[1,i], i);
		(*
		IF(x+1 < 8 AND y+1 < 8 AND NOT GVL.board[x+1,y+1].isEmpty AND GVL.board[x+1,y+1].isBlack) THEN
		
			//possible jump
		END_IF
		*)
		
	END_FOR
	END_IF
END_IF

END_PROGRAM

// Device/Application/clearGlobalStack
FUNCTION clearGlobalStack : bool
VAR_INPUT
END_VAR
VAR
	i : INT := 0;
END_VAR

FOR i := 0 TO 3 DO
	GVL.jumpStack[i].jumpedColor := -1;
	GVL.jumpStack[i].jumpedIndex:= -1;
	GVL.jumpStack[i].xMoveLocation := -1;
	GVL.jumpStack[i].yMoveLocation := -1;
END_FOR

END_FUNCTION

// Device/Application/clearPieceJumpArray
FUNCTION clearPieceJumpArray : BOOL
VAR_INPUT
	pieceColor : INT;
	pieceIndex : INT;
END_VAR
VAR
	i : INT;
END_VAR

FOR i := 0 TO 11 DO
	GVL.pieces[pieceColor,pieceIndex].jumpArr := GVL.emptyJumpArr;
END_FOR

END_FUNCTION

// Device/Application/checkForJumpRed1
FUNCTION checkForJumpRed1 : Piece
VAR_INPUT
	selectedPiece : Piece;
	selectedPieceIndex : INT;
END_VAR

VAR
	i : INT;
	x: INT;
	y: INT;
	xNext : INT;
	yNext : INT;
	jumpedPieceIndex : INT;
	temp : ARRAY [0..1] OF INT;
END_VAR

x := selectedPiece.currentLocation[0];
y := selectedPiece.currentLocation[1];

// checks the board space up and to the right
IF(x+1 < 8 AND y+1 < 8 AND NOT GVL.board[x+1,y+1].isEmpty AND GVL.board[x+1,y+1].isBlack) THEN
	xNext := x + 2; // location of the space you could possibly jump to
	yNext := y + 2; // location of the space you could possibly jump to		
	// if the space that can be jumped to is 
	IF(xNext < 8 AND yNext < 8 AND GVL.board[xNext,yNext].isEmpty) THEN
		selectedPiece.validMoveArr[xNext,yNext] := TRUE;
		temp := findPieceAtGivenLocation(x+1,y+1);
		jumpedPieceIndex := temp[1];
		IF(push(1, jumpedPieceIndex, xNext, yNext)) THEN
			selectedPiece := checkForJumpRed2(selectedPiece, selectedPieceIndex, xNext, yNext);
			selectedPiece := pop(selectedPiece, 0);
		END_IF
	END_IF
END_IF

// checks up and to the left
IF(x-1 >= 0 AND y+1 < 8 AND NOT GVL.board[x-1,y+1].isEmpty AND GVL.board[x-1,y+1].isBlack) THEN
	xNext := x - 2; // location of the space you could possibly jump to
	yNext := y + 2; // location of the space you could possibly jump to
	IF(xNext >= 0 AND yNext < 8 AND GVL.board[xNext,yNext].isEmpty) THEN
		selectedPiece.validMoveArr[xNext,yNext] := TRUE;
		temp := findPieceAtGivenLocation(x-1,y+1);
		jumpedPieceIndex := temp[1];
		IF(push(1, jumpedPieceIndex, xNext, yNext)) THEN
			selectedPiece := checkForJumpRed2(selectedPiece, selectedPieceIndex, xNext, yNext);
			selectedPiece := pop(selectedPiece, 0);
		END_IF
	END_IF
END_IF

checkForJumpRed1 := selectedPiece;


RETURN;

END_FUNCTION

// Device/Application/findPieceAtGivenLocation
FUNCTION findPieceAtGivenLocation : ARRAY[0..1] OF INT
VAR_INPUT
	xLoc : INT;
	yLoc : INT;
END_VAR
VAR
	i : INT;
END_VAR

FOR i := 0 TO 11 DO
	IF(GVL.pieces[0,i].currentLocation[0] = xLoc AND GVL.pieces[0,i].currentLocation[1] = yLoc) THEN
		findPieceAtGivenLocation[0] := 0;
		findPieceAtGivenLocation[1] := i;
	END_IF
	IF(GVL.pieces[1,i].currentLocation[0] = xLoc AND GVL.pieces[1,i].currentLocation[1] = yLoc) THEN
		findPieceAtGivenLocation[0] := 1;
		findPieceAtGivenLocation[1] := i;
	END_IF
END_FOR
RETURN;

END_FUNCTION

// Device/Application/push
FUNCTION push : bool
VAR_INPUT
	jumpedColor : INT;
	jumpedIndex : INT;
	xMoveLoc : INT;
	yMoveLoc : INT;
END_VAR
VAR
	
END_VAR

IF(GVL.currentStackIndex < 4) THEN
	
	// Adds jump information to the current stack
	GVL.jumpStack[GVL.currentStackIndex].xMoveLocation := xMoveLoc;
	GVL.jumpStack[GVL.currentStackIndex].yMoveLocation := yMoveLoc;
	GVL.jumpStack[GVL.currentStackIndex].jumpedColor := jumpedColor;
	GVL.jumpStack[GVL.currentStackIndex].jumpedIndex := jumpedIndex;
	
	// Moves top of the stack up one notch
	GVL.currentStackIndex := GVL.currentStackIndex + 1;
	
	push := TRUE;
ELSE
	// Would indicate that the stack is full (only 4 successive jumps are allowed)
	push := FALSE;
END_IF

END_FUNCTION

// Device/Application/checkForJumpRed2
FUNCTION checkForJumpRed2 : Piece
VAR_INPUT
	selectedPiece : Piece;
	selectedPieceIndex : INT;
	x : INT;
	y : INT;
END_VAR


VAR
	jumpedPieceIndex : INT;
	xNext : INT;
	yNext : INT;
	i : INT;
	temp: ARRAY [0..1] OF INT;
END_VAR

// checks up and to the right
IF(x+1 < 8 AND y+1 < 8 AND NOT GVL.board[x+1,y+1].isEmpty AND GVL.board[x+1,y+1].isBlack) THEN
	xNext := x + 2; // location of the space you could possibly jump to
	yNext := y + 2; // location of the space you could possibly jump to		
	temp := findPieceAtGivenLocation(x+1,y+1);
	selectedPieceIndex := temp[1];
	IF(xNext < 8 AND yNext < 8 AND GVL.board[xNext,yNext].isEmpty) THEN
		selectedPiece.validMoveArr[xNext,yNext] := TRUE;	
		temp := findPieceAtGivenLocation(x+1,y+1);
		jumpedPieceIndex := temp[1];
		IF(push(1, jumpedPieceIndex, xNext, yNext))THEN
			selectedPiece := checkForJumpRed3(selectedPiece, selectedPieceIndex, xNext, yNext);	
			selectedPiece := pop(selectedPiece, 0);
		END_IF
	END_IF
END_IF

// checks up and to the left
IF(x-1 >= 0 AND y+1 < 8 AND NOT GVL.board[x-1,y+1].isEmpty AND GVL.board[x-1,y+1].isBlack) THEN
	xNext := x - 2; // location of the space you could possibly jump to
	yNext := y + 2; // location of the space you could possibly jump to
	IF(xNext >= 0 AND yNext < 8 AND GVL.board[xNext,yNext].isEmpty) THEN
		selectedPiece.validMoveArr[xNext,yNext] := TRUE;
		temp := findPieceAtGivenLocation(x-1,y+1);
		jumpedPieceIndex := temp[1];
		IF(push(1, jumpedPieceIndex, xNext, yNext))THEN
			selectedPiece := checkForJumpRed3(selectedPiece, selectedPieceIndex, xNext, yNext);	
			selectedPiece := pop(selectedPiece, 0);
		END_IF
	END_IF
END_IF

checkForJumpRed2 := selectedPiece;


RETURN;

END_FUNCTION

// Device/Application/checkForJumpRed3
FUNCTION checkForJumpRed3 : Piece
VAR_INPUT
	selectedPiece : Piece;
	selectedPieceIndex : INT;
	x : INT;
	y : INT; 
END_VAR

VAR
	xNext : INT;
	yNext : INT;
	i :INT;
	temp: ARRAY [0..1] OF INT;
	jumpedPieceIndex: INT;
END_VAR

// checks up and to the right
IF(x+1 < 8 AND y+1 < 8 AND NOT GVL.board[x+1,y+1].isEmpty AND GVL.board[x+1,y+1].isBlack) THEN
	xNext := x + 2; // location of the space you could possibly jump to
	yNext := y + 2; // location of the space you could possibly jump to		

	IF(xNext < 8 AND yNext < 8 AND GVL.board[xNext,yNext].isEmpty) THEN
		selectedPiece.validMoveArr[xNext,yNext] := TRUE;
		temp := findPieceAtGivenLocation(x+1,y+1);
		jumpedPieceIndex := temp[1];
		IF(push(1, jumpedPieceIndex, xNext, yNext))THEN
			selectedPiece := checkForJumpRed4(selectedPiece, selectedPieceIndex, xNext, yNext);	
			selectedPiece := pop(selectedPiece, 0);
		END_IF
	END_IF
END_IF

// checks up and to the left
IF(x-1 >= 0 AND y+1 < 8 AND NOT GVL.board[x-1,y+1].isEmpty AND GVL.board[x-1,y+1].isBlack) THEN
	xNext := x - 2; // location of the space you could possibly jump to
	yNext := y + 2; // location of the space you could possibly jump to
	IF(xNext >= 0 AND yNext < 8 AND GVL.board[xNext,yNext].isEmpty) THEN
		selectedPiece.validMoveArr[xNext,yNext] := TRUE;
		temp := findPieceAtGivenLocation(x-1,y+1);
		jumpedPieceIndex := temp[1];
		IF(push(1, jumpedPieceIndex, xNext, yNext))THEN
			selectedPiece := checkForJumpRed4(selectedPiece, selectedPieceIndex, xNext, yNext);	
			selectedPiece := pop(selectedPiece, 0);
		END_IF
	END_IF
END_IF

checkForJumpRed3 := selectedPiece;


RETURN;

END_FUNCTION

// Device/Application/checkForJumpRed4
FUNCTION checkForJumpRed4 : Piece
VAR_INPUT
	selectedPiece : Piece;
	selectedPieceIndex: INT;
	x : INT;
	y : INT; 
END_VAR

VAR
	xNext : INT;
	yNext : INT;
	temp: ARRAY [0..1] OF INT;
	jumpedPieceIndex: INT;
	
END_VAR

// checks up and to the right
IF(x+1 < 8 AND y+1 < 8 AND NOT GVL.board[x+1,y+1].isEmpty AND GVL.board[x+1,y+1].isBlack) THEN
	xNext := x + 2; // location of the space you could possibly jump to
	yNext := y + 2; // location of the space you could possibly jump to		
	IF(xNext < 8 AND yNext < 8 AND GVL.board[xNext,yNext].isEmpty) THEN
		selectedPiece.validMoveArr[xNext,yNext] := TRUE;
		temp := findPieceAtGivenLocation(x+1,y+1);
		jumpedPieceIndex := temp[1];
		IF(push(1, jumpedPieceIndex, xNext, yNext))THEN
			// This is where another jump would be called	
			selectedPiece := pop(selectedPiece, 0);
		END_IF		
	END_IF
END_IF

// checks up and to the left
IF(x-1 >= 0 AND y+1 < 8 AND NOT GVL.board[x-1,y+1].isEmpty AND GVL.board[x-1,y+1].isBlack) THEN
	xNext := x - 2; // location of the space you could possibly jump to
	yNext := y + 2; // location of the space you could possibly jump to
	IF(xNext >= 0 AND yNext < 8 AND GVL.board[xNext,yNext].isEmpty) THEN
		selectedPiece.validMoveArr[xNext,yNext] := TRUE;
		temp := findPieceAtGivenLocation(x-1,y+1);
		jumpedPieceIndex := temp[1];
		IF(push(1, jumpedPieceIndex, xNext, yNext))THEN
			// This is where you would call another jump
			selectedPiece := pop(selectedPiece, 0);
		END_IF	
	
	END_IF
END_IF

checkForJumpRed4 := selectedPiece;


RETURN;

END_FUNCTION

// Device/Application/pop
FUNCTION pop : Piece
VAR_INPUT
	currentPiece : Piece;
	pieceColor : INT;
END_VAR
VAR
	i : INT := 0;
END_VAR

IF(GVL.currentStackIndex = -1) THEN
	// returns false if stack is empty
	pop := currentPiece;
ELSE
	// save the jumpProfile
	FOR i := 0 TO GVL.currentStackIndex - 1 DO
		currentPiece.jumpArr[GVL.currentJumpProfileNum,i].jumpedColor := GVL.jumpStack[i].jumpedColor;
		currentPiece.jumpArr[GVL.currentJumpProfileNum,i].jumpedIndex := GVL.jumpStack[i].jumpedIndex;
		currentPiece.jumpArr[GVL.currentJumpProfileNum,i].xMoveLocation := GVL.jumpStack[i].xMoveLocation;
		currentPiece.jumpArr[GVL.currentJumpProfileNum,i].yMoveLocation := GVL.jumpStack[i].yMoveLocation;
	END_FOR
	
	GVL.currentJumpProfileNum := GVL.currentJumpProfileNum + 1;
	

	// Pops item off of the stack
	GVL.jumpStack[GVL.currentStackIndex].jumpedColor := -1;
	GVL.jumpStack[GVL.currentStackIndex].jumpedIndex := -1;
	GVL.jumpStack[GVL.currentStackIndex].xMoveLocation := -1;
	GVL.jumpStack[GVL.currentStackIndex].yMoveLocation := -1;
	
	// Moves top of stack down
	GVL.currentStackIndex := GVL.currentStackIndex - 1;
	
	pop := currentPiece;
END_IF

RETURN;

END_FUNCTION

// Device/Application/checkForJumpBlack1
FUNCTION checkForJumpBlack1 : Piece
VAR_INPUT
	selectedPiece : Piece;
	selectedPieceIndex : INT;
END_VAR

VAR
	x: INT;
	y: INT;
	i : INT;
	xNext : INT;
	yNext : INT;
	temp: ARRAY [0..1] OF INT;
	jumpedPieceIndex: INT;
END_VAR

x := selectedPiece.currentLocation[0];
y := selectedPiece.currentLocation[1];

// checks down and right
IF(x+1 < 8 AND y-1 >= 0 AND NOT GVL.board[x+1,y-1].isEmpty AND GVL.board[x+1,y-1].isRed) THEN
	xNext := x + 2; // location of the space you could possibly jump to
	yNext := y - 2; // location of the space you could possibly jump to		
	IF(xNext < 8 AND yNext >= 0 AND GVL.board[xNext,yNext].isEmpty) THEN
		selectedPiece.validMoveArr[xNext,yNext] := TRUE;
		temp := findPieceAtGivenLocation(x+1,y-1);
		jumpedPieceIndex := temp[1];
		IF(push(0, jumpedPieceIndex, xNext, yNext)) THEN
			selectedPiece := checkForJumpBlack2(selectedPiece, selectedPieceIndex, xNext, yNext);
			selectedPiece := pop(selectedPiece, 1);
		END_IF
	END_IF
END_IF

// checks down and left
IF(x-1 >= 0 AND y-1 >= 0 AND NOT GVL.board[x-1,y-1].isEmpty AND GVL.board[x-1,y-1].isRed) THEN
	xNext := x - 2; // location of the space you could possibly jump to
	yNext := y - 2; // location of the space you could possibly jump to
	IF(xNext >= 0 AND yNext >= 0 AND GVL.board[xNext,yNext].isEmpty) THEN
		selectedPiece.validMoveArr[xNext,yNext] := TRUE;
		temp := findPieceAtGivenLocation(x-1,y-1);
		jumpedPieceIndex := temp[1];
		IF(push(0, jumpedPieceIndex, xNext, yNext)) THEN
			selectedPiece := checkForJumpBlack2(selectedPiece, selectedPieceIndex, xNext, yNext);
			selectedPiece := pop(selectedPiece, 1);
		END_IF
	END_IF
END_IF

checkForJumpBlack1 := selectedPiece;


RETURN;

END_FUNCTION

// Device/Application/checkForJumpBlack2
FUNCTION checkForJumpBlack2 : Piece
VAR_INPUT
	selectedPiece : Piece;
	selectedPieceIndex : INT;
	x : INT;
	y : INT; 
END_VAR
	
VAR
	i : INT;
	xNext : INT;
	yNext : INT;
	temp: ARRAY [0..1] OF INT;
	jumpedPieceIndex: INT;
END_VAR

// checks down and right
IF(x+1 < 8 AND y-1 >= 0 AND NOT GVL.board[x+1,y-1].isEmpty AND GVL.board[x+1,y-1].isRed) THEN
	xNext := x + 2; // location of the space you could possibly jump to
	yNext := y - 2; // location of the space you could possibly jump to		
	IF(xNext < 8 AND yNext >= 0 AND GVL.board[xNext,yNext].isEmpty) THEN
		selectedPiece.validMoveArr[xNext,yNext] := TRUE;
		temp := findPieceAtGivenLocation(x+1,y-1);
		jumpedPieceIndex := temp[1];
		IF(push(0, jumpedPieceIndex, xNext, yNext)) THEN
			selectedPiece := checkForJumpBlack3(selectedPiece, selectedPieceIndex, xNext, yNext);
			selectedPiece := pop(selectedPiece, 1);
		END_IF
	END_IF
END_IF

// checks down and left
IF(x-1 >= 0 AND y-1 >= 0 AND NOT GVL.board[x-1,y-1].isEmpty AND GVL.board[x-1,y-1].isRed) THEN
	xNext := x - 2; // location of the space you could possibly jump to
	yNext := y - 2; // location of the space you could possibly jump to
	IF(xNext >= 0 AND yNext >= 0 AND GVL.board[xNext,yNext].isEmpty) THEN
		selectedPiece.validMoveArr[xNext,yNext] := TRUE;
		temp := findPieceAtGivenLocation(x-1,y-1);
		jumpedPieceIndex := temp[1];
		IF(push(0, jumpedPieceIndex, xNext, yNext)) THEN
			selectedPiece := checkForJumpBlack3(selectedPiece, selectedPieceIndex, xNext, yNext);
			selectedPiece := pop(selectedPiece, 1);
		END_IF
	END_IF
END_IF

checkForJumpBlack2 := selectedPiece;


RETURN;

END_FUNCTION

// Device/Application/checkForJumpBlack3
FUNCTION checkForJumpBlack3 : Piece
VAR_INPUT
	selectedPiece : Piece;
	selectedPieceIndex : INT;
	x : INT;
	y : INT; 
END_VAR

VAR
	i : INT;
	xNext : INT;
	yNext : INT;
	temp: ARRAY [0..1] OF INT;
	jumpedPieceIndex: INT;
END_VAR

// checks down and right
IF(x+1 < 8 AND y-1 >= 0 AND NOT GVL.board[x+1,y-1].isEmpty AND GVL.board[x+1,y-1].isRed) THEN
	xNext := x + 2; // location of the space you could possibly jump to
	yNext := y - 2; // location of the space you could possibly jump to		
	IF(xNext < 8 AND yNext >= 0 AND GVL.board[xNext,yNext].isEmpty) THEN
		selectedPiece.validMoveArr[xNext,yNext] := TRUE;
		temp := findPieceAtGivenLocation(x+1,y-1);
		jumpedPieceIndex := temp[1];
		IF(push(0, jumpedPieceIndex, xNext, yNext)) THEN
			selectedPiece := checkForJumpBlack4(selectedPiece, selectedPieceIndex, xNext, yNext);
			selectedPiece := pop(selectedPiece, 1);
		END_IF
	END_IF
END_IF

// checks down and left
IF(x-1 >= 0 AND y-1 >= 0 AND NOT GVL.board[x-1,y-1].isEmpty AND GVL.board[x-1,y-1].isRed) THEN
	xNext := x - 2; // location of the space you could possibly jump to
	yNext := y - 2; // location of the space you could possibly jump to
	IF(xNext >= 0 AND yNext >= 0 AND GVL.board[xNext,yNext].isEmpty) THEN
		selectedPiece.validMoveArr[xNext,yNext] := TRUE;
		temp := findPieceAtGivenLocation(x-1,y-1);
		jumpedPieceIndex := temp[1];
		IF(push(0, jumpedPieceIndex, xNext, yNext)) THEN
			selectedPiece := checkForJumpBlack4(selectedPiece, selectedPieceIndex, xNext, yNext);
			selectedPiece := pop(selectedPiece, 1);
		END_IF		
	END_IF
END_IF

checkForJumpBlack3 := selectedPiece;


RETURN;

END_FUNCTION

// Device/Application/checkForJumpBlack4
FUNCTION checkForJumpBlack4 : Piece
VAR_INPUT
	selectedPiece : Piece;
	selectedPieceIndex : INT;
	x : INT;
	y : INT; 
END_VAR

VAR
	xNext : INT;
	yNext : INT;
	temp: ARRAY [0..1] OF INT;
	jumpedPieceIndex: INT;
END_VAR

// checks down and right
IF(x+1 < 8 AND y-1 >= 0 AND NOT GVL.board[x+1,y-1].isEmpty AND GVL.board[x+1,y-1].isRed) THEN
	xNext := x + 2; // location of the space you could possibly jump to
	yNext := y - 2; // location of the space you could possibly jump to		
	IF(xNext < 8 AND yNext >= 0 AND GVL.board[xNext,yNext].isEmpty) THEN
		selectedPiece.validMoveArr[xNext,yNext] := TRUE;
		temp := findPieceAtGivenLocation(x+1,y-1);
		jumpedPieceIndex := temp[1];
		IF(push(0, jumpedPieceIndex, xNext, yNext)) THEN
			//selectedPiece := checkForJumpBlack2(selectedPiece, selectedPieceIndex, xNext, yNext);
			selectedPiece := pop(selectedPiece, 1);
		END_IF
	END_IF
END_IF

// checks down and left
IF(x-1 >= 0 AND y-1 >= 0 AND NOT GVL.board[x-1,y-1].isEmpty AND GVL.board[x-1,y-1].isRed) THEN
	xNext := x - 2; // location of the space you could possibly jump to
	yNext := y - 2; // location of the space you could possibly jump to
	IF(xNext >= 0 AND yNext >= 0 AND GVL.board[xNext,yNext].isEmpty) THEN
		selectedPiece.validMoveArr[xNext,yNext] := TRUE;
		temp := findPieceAtGivenLocation(x-1,y-1);
		jumpedPieceIndex := temp[1];
		IF(push(0, jumpedPieceIndex, xNext, yNext)) THEN
			//selectedPiece := checkForJumpBlack2(selectedPiece, selectedPieceIndex, xNext, yNext);
			selectedPiece := pop(selectedPiece, 1);
		END_IF
	END_IF
END_IF

checkForJumpBlack4 := selectedPiece;


RETURN;

END_FUNCTION

// Device/Application/ClearTakenPieces
PROGRAM ClearTakenPieces
VAR
	i : INT := 99;
	j : INT;
	k : INT;
	t : INT;
	currentRef : INT;
	found : BOOL;
END_VAR

IF(GVL.xMoveSpace <> -1 AND GVL.yMoveSpace <> -1) THEN
	i := 30;
	found := FALSE;
	WHILE(i >= 0 AND NOT found) DO
		
		
		// If the space identified in the jump move array and the space chosen match
		IF(GVL.jumpMoveArr[i].xMoveLocation = GVL.xMoveSpace AND GVL.jumpMoveArr[i].yMoveLocation = GVL.yMoveSpace) THEN
			found := TRUE;
			j := GVL.jumpMoveArr[i].jumpRef;
			k := i;
			WHILE(j >= 0 AND k >= 0) DO
				IF(GVL.jumpMoveArr[k].jumpRef = j) THEN					
					// Moves piece to its original location (off of the board)
					GVL.pieces[GVL.jumpMoveArr[k].jumpedPieceColor, GVL.jumpMoveArr[k].jumpedPieceIndex].translatedLocation[0] := 0;
					GVL.pieces[GVL.jumpMoveArr[k].jumpedPieceColor, GVL.jumpMoveArr[k].jumpedPieceIndex].translatedLocation[1] := 0;
						
					// Nulls out information for all taken pieces
					GVL.pieces[GVL.jumpMoveArr[k].jumpedPieceColor, GVL.jumpMoveArr[k].jumpedPieceIndex].isTaken := TRUE;	
					GVL.pieces[GVL.jumpMoveArr[k].jumpedPieceColor, GVL.jumpMoveArr[k].jumpedPieceIndex].isKing := FALSE;
					
					IF(GVL.board[GVL.jumpMoveArr[k].xJumpedLocation, GVL.jumpMoveArr[k].yJumpedLocation].isBlack) THEN
						GVL.blackPiecesTaken := GVL.blackPiecesTaken + 1;
					END_IF
					
					// Clears board space occupied by piece that was jumped
					GVL.board[GVL.jumpMoveArr[k].xJumpedLocation, GVL.jumpMoveArr[k].yJumpedLocation].isEmpty := TRUE;
					GVL.board[GVL.jumpMoveArr[k].xJumpedLocation, GVL.jumpMoveArr[k].yJumpedLocation].isRed := FALSE;
					GVL.board[GVL.jumpMoveArr[k].xJumpedLocation, GVL.jumpMoveArr[k].yJumpedLocation].isBlack := FALSE;
					
						
					// Sets pieces current location to invalid values
					GVL.pieces[GVL.jumpMoveArr[k].jumpedPieceColor, GVL.jumpMoveArr[k].jumpedPieceIndex].currentLocation[0] := -1;
					GVL.pieces[GVL.jumpMoveArr[k].jumpedPieceColor, GVL.jumpMoveArr[k].jumpedPieceIndex].currentLocation[1] := -1;
						
					// Nulls out pieces current valid move array
					GVL.pieces[GVL.jumpMoveArr[k].jumpedPieceColor, GVL.jumpMoveArr[k].jumpedPieceIndex].validMoveArr := GVL.noValidMoveArr;
					
					j := GVL.jumpMoveArr[k].lastJumpRef;
					
					WHILE(GVL.test) DO
								//
					END_WHILE
					
				END_IF
				k := k - 1;
			END_WHILE
		END_IF
		i := i - 1;
	END_WHILE
	(*FOR i := 0 TO 8 DO
		GVL.jumpMoveArr[i].numPiecesToJump := 0;
		GVL.jumpMoveArr[i].jumpedPieceColor := 0;
		GVL.jumpMoveArr[i].jumpedPieceIndex := 0;
		GVL.jumpMoveArr[i].xMoveLocation := 0;
		GVL.jumpMoveArr[i].yMoveLocation := 0;
	END_FOR*)
END_IF

END_PROGRAM

// Device/Application/clearJumpArr
FUNCTION clearJumpArr : Bool
VAR_INPUT
END_VAR
VAR
	i : INT;
END_VAR

FOR i := 0 TO 99 DO
	GVL.jumpMoveArr[i].jumpedPieceColor := 0;
	GVL.jumpMoveArr[i].jumpedPieceIndex := 0;
	GVL.jumpMoveArr[i].jumpRef := 0;
	GVL.jumpMoveArr[i].lastJumpRef := -1;
	GVL.jumpMoveArr[i].numPiecesToJump := 0;
	GVL.jumpMoveArr[i].xJumpedLocation := 0;
	GVL.jumpMoveArr[i].xMoveLocation := 0;
	GVL.jumpMoveArr[i].yJumpedLocation := 0;
	GVL.jumpMoveArr[i].yMoveLocation := 0;
END_FOR

RETURN;

END_FUNCTION

// Device/Application/MovePieceMotion
FUNCTION_BLOCK MovePieceMotion
VAR_INPUT
	xPos: LREAL;
	yPos: LREAL;
	zPos: LREAL;
	ExecuteMove: BOOL;
END_VAR
VAR_IN_OUT
	AxisGroup: AXIS_GROUP_REF_SM3;
END_VAR

VAR_OUTPUT
	
	MoveDone: BOOL;
END_VAR
VAR
	MoveCommand: MC_MoveDirectAbsolute;
	
END_VAR
VAR // added by the converter: edge detectors and wires of the graphical bodies
    _s1 : MC_COORD_REF;
    _s2 : SMC_POS_REF;
END_VAR

// compose _s1 : MC_COORD_REF
_s1.X := xPos;
_s1.Y := yPos;
_s1.Z := zPos;
MoveCommand(
    AxisGroup := AxisGroup,
    Execute := ExecuteMove,
    Position := _s2,
    CoordSystem := SMC_COORD_SYSTEM.MCS,
    BufferMode := MC_BUFFER_MODE.Buffered,
    VelFactor := 1,
    AccFactor := 1,
    JerkFactor := 1); // MC_MoveDirectAbsolute
MoveDone := MoveCommand.Done;
// compose _s2 : SMC_POS_REF
_s2.c := _s1;

END_FUNCTION_BLOCK

// Device/Application/timeDelay
FUNCTION_BLOCK timeDelay
VAR_INPUT
	startTimer: BOOL;
END_VAR
VAR_OUTPUT
	done : BOOL;
END_VAR
VAR
	TON_0: TON;
END_VAR

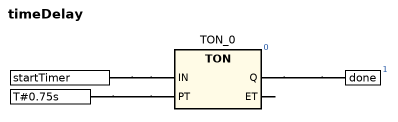
TON_0(IN := startTimer, PT := T#0.75s); // TON
done := TON_0.Q;

END_FUNCTION_BLOCK

// Device/Application/AxisPositionFeedback
PROGRAM AxisPositionFeedback
VAR
	ReadPos: MC_GroupReadActualPosition;
	pos: SMC_POS_REF;
	enable: BOOL;
END_VAR

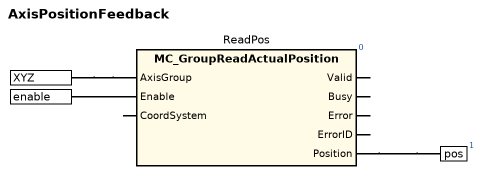
ReadPos(AxisGroup := XYZ, Enable := enable); // MC_GroupReadActualPosition
pos := ReadPos.Position;

END_PROGRAM

// Device/Application/HMISequence
PROGRAM HMISequence
VAR
END_VAR

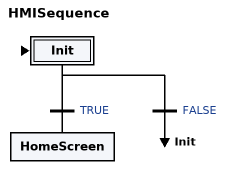
INITIAL_STEP Init:
END_STEP
TRANSITION FROM Init TO HomeScreen
    := TRUE;
END_TRANSITION
TRANSITION FROM Init TO Init
    := FALSE;
END_TRANSITION
STEP HomeScreen:
END_STEP

END_PROGRAM

// Device/Application/placePiece
FUNCTION placePiece : ARRAY [0..1] OF INT

VAR_INPUT
	isBlack : BOOL;
	pieceNum : INT;
END_VAR
VAR
	x : INT;
	y : INT;
	temp : INT;
END_VAR

// Set up for black
IF(isBlack) THEN
	y := pieceNum / 4;
	x := ((2 * pieceNum) MOD 8) + (y MOD 2);
// Setup for red
ELSE
	temp := pieceNum / 4;
	y := temp + 5;
	x := (((2 * pieceNum) MOD 8) + (temp MOD 2)) + 1;
	IF(x >= 8) THEN
		x := 0;
	END_IF
END_IF

placePiece[0] := x;
placePiece[1] := y;

RETURN;

END_FUNCTION

// Device/Application/ProgramFlow
PROGRAM ProgramFlow
VAR
	PlayGame: BOOL;
END_VAR
// where we displace player move options?

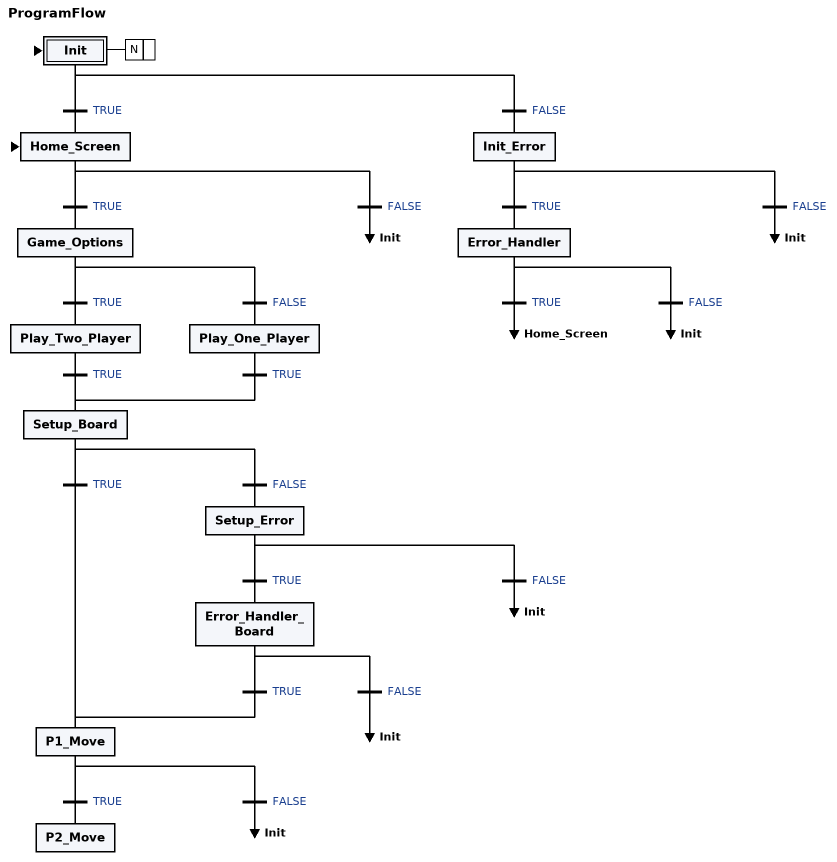
INITIAL_STEP Init:
    // ???(N);
END_STEP
TRANSITION FROM Init TO Home_Screen
    := TRUE;
END_TRANSITION
TRANSITION FROM Init TO Init_Error
    := FALSE;
END_TRANSITION
STEP Init_Error:
END_STEP
TRANSITION FROM Init_Error TO Error_Handler
    := TRUE;
END_TRANSITION
STEP Error_Handler:
END_STEP
TRANSITION FROM Error_Handler TO Home_Screen
    := TRUE;
END_TRANSITION
TRANSITION FROM Error_Handler TO Init
    := FALSE;
END_TRANSITION
TRANSITION FROM Init_Error TO Init
    := FALSE;
END_TRANSITION
STEP Home_Screen:
END_STEP
TRANSITION FROM Home_Screen TO Game_Options
    := TRUE;
END_TRANSITION
TRANSITION FROM Home_Screen TO Init
    := FALSE;
END_TRANSITION
STEP Game_Options:
END_STEP
TRANSITION FROM Game_Options TO Play_Two_Player
    := TRUE;
END_TRANSITION
STEP Play_Two_Player:
END_STEP
TRANSITION FROM Play_Two_Player TO Setup_Board
    := TRUE;
END_TRANSITION
TRANSITION FROM Game_Options TO Play_One_Player
    := FALSE;
END_TRANSITION
STEP Play_One_Player:
END_STEP
TRANSITION FROM Play_One_Player TO Setup_Board
    := TRUE;
END_TRANSITION
STEP Setup_Board:
END_STEP
TRANSITION FROM Setup_Board TO P1_Move
    := TRUE;
END_TRANSITION
TRANSITION FROM Setup_Board TO Setup_Error
    := FALSE;
END_TRANSITION
STEP Setup_Error:
END_STEP
TRANSITION FROM Setup_Error TO Error_Handler_Board
    := TRUE;
END_TRANSITION
TRANSITION FROM Setup_Error TO Init
    := FALSE;
END_TRANSITION
STEP Error_Handler_Board:
END_STEP
TRANSITION FROM Error_Handler_Board TO P1_Move
    := TRUE;
END_TRANSITION
TRANSITION FROM Error_Handler_Board TO Init
    := FALSE;
END_TRANSITION
STEP P1_Move:
END_STEP
TRANSITION FROM P1_Move TO P2_Move
    := TRUE;
END_TRANSITION
TRANSITION FROM P1_Move TO Init
    := FALSE;
END_TRANSITION
STEP P2_Move:
END_STEP

END_PROGRAM

// Device/Application/Init
PROGRAM Init
VAR
END_VAR

END_PROGRAM

// Device/Application/movePiece
FUNCTION movePiece : Piece
VAR_INPUT
	currentPiece : Piece;
	spaceX : INT; // space that you the user wants to move to
	spaceY : INT; // space that the user wants to move to
END_VAR
VAR
	spaceTranslation : ARRAY [0..1] OF INT; // small numbers (0-7) that indicate how many spaces a piece needs to be moved
	sizeOfMoveX : INT := 50;
	sizeOfMoveY : INT := -50;
END_VAR

// DOESN'T DO ANYTHING, DEPRECATE


IF(currentPiece.validMoveArr[spaceX, spaceY]) THEN
	
	// Tells you how many spaces you need to move
	spaceTranslation[0] := spaceX - currentPiece.currentLocation[0];
	spaceTranslation[1] := spaceY - currentPiece.currentLocation[1];

	// Converts spaces needed to move into pixels needed to move
	currentPiece.translatedLocation[0] := spaceTranslation[0] * sizeOfMoveX;
	currentPiece.translatedLocation[1] := spaceTranslation[1] * sizeOfMoveY;
	
	// sets old location to the current location
	currentPiece.oldLocation[0] := currentPiece.currentLocation[0];
	currentPiece.oldLocation[1] := currentPiece.currentLocation[1];
	
	// updates the current location
	currentPiece.currentLocation[0] := spaceX;
	currentPiece.currentLocation[1] := spaceY;
	
END_IF

movePiece := currentPiece;
currentPiece.isSelected := FALSE;

RETURN;

END_FUNCTION

// Device/Application/pieceSelect
FUNCTION pieceSelect : ARRAY[0..1,0..11] OF Piece;
VAR_INPUT
	pieces : ARRAY[0..1,0..11] OF Piece;
	selectedPieceValidMoveArr : ARRAY[0..7,0..7] OF BOOL;
END_VAR
VAR
	i :INT;
END_VAR

FOR i := 0 TO 11 DO
	pieces[0,i].isSelected := FALSE;
	pieces[1,i].isSelected := FALSE;
END_FOR

selectedPieceValidMoveArr := pieces[0,10].validMoveArr;
pieceSelect := pieces;

END_FUNCTION

// Device/Application/JumpPieces
PROGRAM JumpPieces
VAR
	i : INT;
	selectedPieceColor : INT;
	selectedPieceIndex : INT;
END_VAR

END_PROGRAM

// Device/Application/Loading_Screen
VISUALIZATION Loading_Screen  // 2x2
END_VISUALIZATION

// Device/Application/Home_Screen
VISUALIZATION Home_Screen  // 2x2
END_VISUALIZATION

// Device/Application/Checkerboard
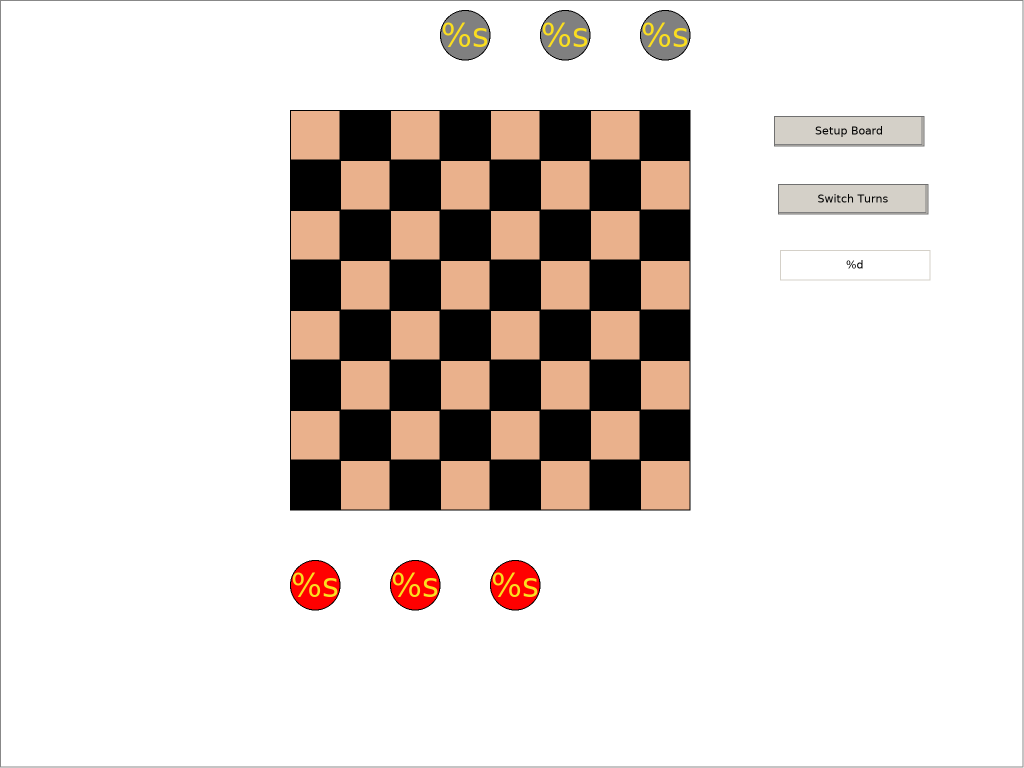
VISUALIZATION Checkerboard  // 1024x768
VAR_IN_OUT
	
END_VAR

VAR
	i : INT;
END_VAR
    Rectangle (290,260 50x50), colour toggle: GVL.selectedPieceValidMoveArr[0,4]
        OnMouseClick: execute { GVL.xMoveSpace := 0; GVL.yMoveSpace := 4; }
    Rectangle (340,260 50x50)
    Rectangle (390,260 50x50), colour toggle: GVL.selectedPieceValidMoveArr[2,4]
        OnMouseClick: execute { GVL.xMoveSpace := 2; GVL.yMoveSpace := 4; }
    Rectangle (440,260 50x50)
    Rectangle (290,210 50x50)
    Rectangle (340,210 50x50), colour toggle: GVL.selectedPieceValidMoveArr[1,5]
        OnMouseClick: execute { GVL.xMoveSpace := 1; GVL.yMoveSpace := 5; }
    Rectangle (390,210 50x50)
    Rectangle (440,210 50x50), colour toggle: GVL.selectedPieceValidMoveArr[3,5]
        OnMouseClick: execute { GVL.xMoveSpace := 3; GVL.yMoveSpace := 5; }
    Rectangle (290,160 50x50), colour toggle: GVL.selectedPieceValidMoveArr[0,6]
        OnMouseClick: execute { GVL.xMoveSpace := 0; GVL.yMoveSpace := 6; }
    Rectangle (340,160 50x50)
    Rectangle (390,160 50x50), colour toggle: GVL.selectedPieceValidMoveArr[2,6]
        OnMouseClick: execute { GVL.xMoveSpace := 2; GVL.yMoveSpace := 6; }
    Rectangle (440,160 50x50)
    Rectangle (290,110 50x50)
    Rectangle (440,110 50x50), colour toggle: GVL.selectedPieceValidMoveArr[3,7]
        OnMouseClick: execute { GVL.xMoveSpace := 3; GVL.yMoveSpace := 7; }
    Rectangle (390,110 50x50)
    Rectangle (340,110 50x50), colour toggle: GVL.selectedPieceValidMoveArr[1,7]
        OnMouseClick: execute { GVL.xMoveSpace := 1; GVL.yMoveSpace := 7; }
    Rectangle (490,260 50x50), colour toggle: GVL.selectedPieceValidMoveArr[4,4]
        OnMouseClick: execute { GVL.xMoveSpace := 4; GVL.yMoveSpace := 4; }
    Rectangle (540,260 50x50)
    Rectangle (590,260 50x50), colour toggle: GVL.selectedPieceValidMoveArr[6,4]
        OnMouseClick: execute { GVL.xMoveSpace := 6; GVL.yMoveSpace := 4; }
    Rectangle (640,260 50x50)
    Rectangle (490,210 50x50)
    Rectangle (540,210 50x50), colour toggle: GVL.selectedPieceValidMoveArr[5,5]
        OnMouseClick: execute { GVL.xMoveSpace := 5; GVL.yMoveSpace := 5; }
    Rectangle (590,210 50x50)
    Rectangle (640,210 50x50), colour toggle: GVL.selectedPieceValidMoveArr[7,5]
        OnMouseClick: execute { GVL.xMoveSpace := 7; GVL.yMoveSpace := 5; }
    Rectangle (490,160 50x50), colour toggle: GVL.selectedPieceValidMoveArr[4,6]
        OnMouseClick: execute { GVL.xMoveSpace := 4; GVL.yMoveSpace := 6; }
    Rectangle (540,160 50x50)
    Rectangle (590,160 50x50), colour toggle: GVL.selectedPieceValidMoveArr[6,6]
        OnMouseClick: execute { GVL.xMoveSpace := 6; GVL.yMoveSpace := 6; }
    Rectangle (640,160 50x50)
    Rectangle (490,110 50x50)
    Rectangle (640,110 50x50), colour toggle: GVL.selectedPieceValidMoveArr[7,7]
        OnMouseClick: execute { GVL.xMoveSpace := 7; GVL.yMoveSpace := 7; }
    Rectangle (590,110 50x50)
    Rectangle (540,110 50x50), colour toggle: GVL.selectedPieceValidMoveArr[5,7]
        OnMouseClick: execute { GVL.xMoveSpace := 5; GVL.yMoveSpace := 7; }
    Rectangle (490,460 50x50), colour toggle: GVL.selectedPieceValidMoveArr[4,0]
        OnMouseClick: execute { GVL.xMoveSpace := 4; GVL.yMoveSpace := 0; }
    Rectangle (540,460 50x50)
    Rectangle (590,460 50x50), colour toggle: GVL.selectedPieceValidMoveArr[6,0]
        OnMouseClick: execute { GVL.xMoveSpace := 6; GVL.yMoveSpace := 0; }
    Rectangle (640,460 50x50)
    Rectangle (490,410 50x50)
    Rectangle (540,410 50x50), colour toggle: GVL.selectedPieceValidMoveArr[5,1]
        OnMouseClick: execute { GVL.xMoveSpace := 5; GVL.yMoveSpace := 1; }
    Rectangle (590,410 50x50)
    Rectangle (640,410 50x50), colour toggle: GVL.selectedPieceValidMoveArr[7,1]
        OnMouseClick: execute { GVL.xMoveSpace := 7; GVL.yMoveSpace := 1; }
    Rectangle (490,360 50x50), colour toggle: GVL.selectedPieceValidMoveArr[4,2]
        OnMouseClick: execute { GVL.xMoveSpace := 4; GVL.yMoveSpace := 2; }
    Rectangle (540,360 50x50)
    Rectangle (590,360 50x50), colour toggle: GVL.selectedPieceValidMoveArr[6,2]
        OnMouseClick: execute { GVL.xMoveSpace := 6; GVL.yMoveSpace := 2; }
    Rectangle (640,360 50x50)
    Rectangle (490,310 50x50)
    Rectangle (640,310 50x50), colour toggle: GVL.selectedPieceValidMoveArr[7,3]
        OnMouseClick: execute { GVL.xMoveSpace := 7; GVL.yMoveSpace := 3; }
    Rectangle (590,310 50x50)
    Rectangle (540,310 50x50), colour toggle: GVL.selectedPieceValidMoveArr[5,3]
        OnMouseClick: execute { GVL.xMoveSpace := 5; GVL.yMoveSpace := 3; }
    Rectangle (290,460 50x50), colour toggle: GVL.selectedPieceValidMoveArr[0,0]
        OnMouseClick: execute { GVL.xMoveSpace := 0; GVL.yMoveSpace := 0; }
    Rectangle (340,460 50x50)
    Rectangle (390,460 50x50), colour toggle: GVL.selectedPieceValidMoveArr[2,0]
        OnMouseClick: execute { GVL.xMoveSpace := 2; GVL.yMoveSpace := 0; }
    Rectangle (440,460 50x50)
    Rectangle (290,410 50x50)
    Rectangle (340,410 50x50), colour toggle: GVL.selectedPieceValidMoveArr[1,1]
        OnMouseClick: execute { GVL.xMoveSpace := 1; GVL.yMoveSpace := 1; }
    Rectangle (390,410 50x50)
    Rectangle (440,410 50x50), colour toggle: GVL.selectedPieceValidMoveArr[3,1]
        OnMouseClick: execute { GVL.xMoveSpace := 3; GVL.yMoveSpace := 1; }
    Rectangle (290,360 50x50), colour toggle: GVL.selectedPieceValidMoveArr[0,2]
        OnMouseClick: execute { GVL.xMoveSpace := 0; GVL.yMoveSpace := 2; }
    Rectangle (340,360 50x50)
    Rectangle (390,360 50x50), colour toggle: GVL.selectedPieceValidMoveArr[2,2]
        OnMouseClick: execute { GVL.xMoveSpace := 2; GVL.yMoveSpace := 2; }
    Rectangle (440,360 50x50)
    Rectangle (290,310 50x50)
    Rectangle (440,310 50x50), colour toggle: GVL.selectedPieceValidMoveArr[3,3]
        OnMouseClick: execute { GVL.xMoveSpace := 3; GVL.yMoveSpace := 3; }
    Rectangle (390,310 50x50)
    Rectangle (340,310 50x50), colour toggle: GVL.selectedPieceValidMoveArr[1,3]
        OnMouseClick: execute { GVL.xMoveSpace := 1; GVL.yMoveSpace := 3; }
    Ellipse (490,560 50x50), "%s", text variable: GVL.pieces[0,11].kingText, colour toggle: GVL.pieces[0,11].isSelected
        p3560616238: GVL.pieces[0,11].translatedLocation[0]
        p2738717112: GVL.pieces[0,11].translatedLocation[1]
        OnMouseClick: execute {
            IF(NOT GVL.pieces[0,11].isSelected) THEN
            	// deselect everything
            	FOR i := 0 TO 11 DO
            		GVL.pieces[0,i].isSelected := FALSE;
            		GVL.pieces[1,i].isSelected := FALSE;
            	END_FOR
            	// select the piece
            	GVL.pieces[0,11].isSelected := TRUE;
            	GVL.selectedPieceValidMoveArr := GVL.pieces[0,11].validMoveArr;
            ELSE
            	GVL.pieces[0,11].isSelected := FALSE;
            	GVL.selectedPieceValidMoveArr := GVL.noValidMoveArr;
            END_IF
        }
    Ellipse (490,560 50x50), "%s", text variable: GVL.pieces[0,10].kingText, colour toggle: GVL.pieces[0,10].isSelected
        p3560616238: GVL.pieces[0,10].translatedLocation[0]
        p2738717112: GVL.pieces[0,10].translatedLocation[1]
        OnMouseClick: execute {
            IF(NOT GVL.pieces[0,10].isSelected) THEN
            	// deselect everything
            	FOR i := 0 TO 11 DO
            		GVL.pieces[0,i].isSelected := FALSE;
            		GVL.pieces[1,i].isSelected := FALSE;
            	END_FOR
            	// select the piece
            	GVL.pieces[0,10].isSelected := TRUE;
            	GVL.selectedPieceValidMoveArr := GVL.pieces[0,10].validMoveArr;
            ELSE
            	GVL.pieces[0,10].isSelected := FALSE;
            	GVL.selectedPieceValidMoveArr := GVL.noValidMoveArr;
            END_IF
        }
    Ellipse (390,560 50x50), "%s", text variable: GVL.pieces[0,9].kingText, colour toggle: GVL.pieces[0,9].isSelected
        p3560616238: GVL.pieces[0,9].translatedLocation[0]
        p2738717112: GVL.pieces[0,9].translatedLocation[1]
        OnMouseClick: execute {
            IF(NOT GVL.pieces[0,9].isSelected) THEN
            	// deselect everything
            	FOR i := 0 TO 11 DO
            		GVL.pieces[0,i].isSelected := FALSE;
            		GVL.pieces[1,i].isSelected := FALSE;
            	END_FOR
            	// select the piece
            	GVL.pieces[0,9].isSelected := TRUE;
            	GVL.selectedPieceValidMoveArr := GVL.pieces[0,9].validMoveArr;
            ELSE
            	GVL.pieces[0,9].isSelected := FALSE;
            	GVL.selectedPieceValidMoveArr := GVL.noValidMoveArr;
            END_IF
        }
    Ellipse (390,560 50x50), "%s", text variable: GVL.pieces[0,8].kingText, colour toggle: GVL.pieces[0,8].isSelected
        p3560616238: GVL.pieces[0,8].translatedLocation[0]
        p2738717112: GVL.pieces[0,8].translatedLocation[1]
        OnMouseClick: execute {
            IF(NOT GVL.pieces[0,8].isSelected) THEN
            	// deselect everything
            	FOR i := 0 TO 11 DO
            		GVL.pieces[0,i].isSelected := FALSE;
            		GVL.pieces[1,i].isSelected := FALSE;
            	END_FOR
            	// select the piece
            	GVL.pieces[0,8].isSelected := TRUE;
            	GVL.selectedPieceValidMoveArr := GVL.pieces[0,8].validMoveArr;
            ELSE
            	GVL.pieces[0,8].isSelected := FALSE;
            	GVL.selectedPieceValidMoveArr := GVL.noValidMoveArr;
            END_IF
        }
    Ellipse (390,560 50x50), "%s", text variable: GVL.pieces[0,7].kingText, colour toggle: GVL.pieces[0,7].isSelected
        p3560616238: GVL.pieces[0,7].translatedLocation[0]
        p2738717112: GVL.pieces[0,7].translatedLocation[1]
        OnMouseClick: execute {
            IF(NOT GVL.pieces[0,7].isSelected) THEN
            	// deselect everything
            	FOR i := 0 TO 11 DO
            		GVL.pieces[0,i].isSelected := FALSE;
            		GVL.pieces[1,i].isSelected := FALSE;
            	END_FOR
            	// select the piece
            	GVL.pieces[0,7].isSelected := TRUE;
            	GVL.selectedPieceValidMoveArr := GVL.pieces[0,7].validMoveArr;
            ELSE
            	GVL.pieces[0,7].isSelected := FALSE;
            	GVL.selectedPieceValidMoveArr := GVL.noValidMoveArr;
            END_IF
        }
    Ellipse (390,560 50x50), "%s", text variable: GVL.pieces[0,6].kingText, colour toggle: GVL.pieces[0,6].isSelected
        p3560616238: GVL.pieces[0,6].translatedLocation[0]
        p2738717112: GVL.pieces[0,6].translatedLocation[1]
        OnMouseClick: execute {
            IF(NOT GVL.pieces[0,6].isSelected) THEN
            	// deselect everything
            	FOR i := 0 TO 11 DO
            		GVL.pieces[0,i].isSelected := FALSE;
            		GVL.pieces[1,i].isSelected := FALSE;
            	END_FOR
            	// select the piece
            	GVL.pieces[0,6].isSelected := TRUE;
            	GVL.selectedPieceValidMoveArr := GVL.pieces[0,6].validMoveArr;
            ELSE
            	GVL.pieces[0,6].isSelected := FALSE;
            	GVL.selectedPieceValidMoveArr := GVL.noValidMoveArr;
            END_IF
        }
    Ellipse (390,560 50x50), "%s", text variable: GVL.pieces[0,5].kingText, colour toggle: GVL.pieces[0,5].isSelected
        p3560616238: GVL.pieces[0,5].translatedLocation[0]
        p2738717112: GVL.pieces[0,5].translatedLocation[1]
        OnMouseClick: execute {
            IF(NOT GVL.pieces[0,5].isSelected) THEN
            	// deselect everything
            	FOR i := 0 TO 11 DO
            		GVL.pieces[0,i].isSelected := FALSE;
            		GVL.pieces[1,i].isSelected := FALSE;
            	END_FOR
            	// select the piece
            	GVL.pieces[0,5].isSelected := TRUE;
            	GVL.selectedPieceValidMoveArr := GVL.pieces[0,5].validMoveArr;
            ELSE
            	GVL.pieces[0,5].isSelected := FALSE;
            	GVL.selectedPieceValidMoveArr := GVL.noValidMoveArr;
            END_IF
        }
    Ellipse (290,560 50x50), "%s", text variable: GVL.pieces[0,4].kingText, colour toggle: GVL.pieces[0,4].isSelected
        p3560616238: GVL.pieces[0,4].translatedLocation[0]
        p2738717112: GVL.pieces[0,4].translatedLocation[1]
        OnMouseClick: execute {
            IF(NOT GVL.pieces[0,4].isSelected) THEN
            	// deselect everything
            	FOR i := 0 TO 11 DO
            		GVL.pieces[0,i].isSelected := FALSE;
            		GVL.pieces[1,i].isSelected := FALSE;
            	END_FOR
            	// select the piece
            	GVL.pieces[0,4].isSelected := TRUE;
            	GVL.selectedPieceValidMoveArr := GVL.pieces[0,4].validMoveArr;
            ELSE
            	GVL.pieces[0,4].isSelected := FALSE;
            	GVL.selectedPieceValidMoveArr := GVL.noValidMoveArr;
            END_IF
        }
    Ellipse (290,560 50x50), "%s", text variable: GVL.pieces[0,3].kingText, colour toggle: GVL.pieces[0,3].isSelected
        p3560616238: GVL.pieces[0,3].translatedLocation[0]
        p2738717112: GVL.pieces[0,3].translatedLocation[1]
        OnMouseClick: execute {
            IF(NOT GVL.pieces[0,3].isSelected) THEN
            	// deselect everything
            	FOR i := 0 TO 11 DO
            		GVL.pieces[0,i].isSelected := FALSE;
            		GVL.pieces[1,i].isSelected := FALSE;
            	END_FOR
            	// select the piece
            	GVL.pieces[0,3].isSelected := TRUE;
            	GVL.selectedPieceValidMoveArr := GVL.pieces[0,3].validMoveArr;
            ELSE
            	GVL.pieces[0,3].isSelected := FALSE;
            	GVL.selectedPieceValidMoveArr := GVL.noValidMoveArr;
            END_IF
        }
    Ellipse (290,560 50x50), "%s", text variable: GVL.pieces[0,2].kingText, colour toggle: GVL.pieces[0,2].isSelected
        p3560616238: GVL.pieces[0,2].translatedLocation[0]
        p2738717112: GVL.pieces[0,2].translatedLocation[1]
        OnMouseClick: execute {
            IF(NOT GVL.pieces[0,2].isSelected) THEN
            	// deselect everything
            	FOR i := 0 TO 11 DO
            		GVL.pieces[0,i].isSelected := FALSE;
            		GVL.pieces[1,i].isSelected := FALSE;
            	END_FOR
            	// select the piece
            	GVL.pieces[0,2].isSelected := TRUE;
            	GVL.selectedPieceValidMoveArr := GVL.pieces[0,2].validMoveArr;
            ELSE
            	GVL.pieces[0,2].isSelected := FALSE;
            	GVL.selectedPieceValidMoveArr := GVL.noValidMoveArr;
            END_IF
        }
    Ellipse (290,560 50x50), "%s", text variable: GVL.pieces[0,1].kingText, colour toggle: GVL.pieces[0,1].isSelected
        p3560616238: GVL.pieces[0,1].translatedLocation[0]
        p2738717112: GVL.pieces[0,1].translatedLocation[1]
        OnMouseClick: execute {
            IF(NOT GVL.pieces[0,1].isSelected) THEN
            	// deselect everything
            	FOR i := 0 TO 11 DO
            		GVL.pieces[0,i].isSelected := FALSE;
            		GVL.pieces[1,i].isSelected := FALSE;
            	END_FOR
            	// select the piece
            	GVL.pieces[0,1].isSelected := TRUE;
            	GVL.selectedPieceValidMoveArr := GVL.pieces[0,1].validMoveArr;
            ELSE
            	GVL.pieces[0,1].isSelected := FALSE;
            	GVL.selectedPieceValidMoveArr := GVL.noValidMoveArr;
            END_IF
        }
    Ellipse (290,560 50x50), "%s", text variable: GVL.pieces[0,0].kingText, colour toggle: GVL.pieces[0,0].isSelected
        p3560616238: GVL.pieces[0,0].translatedLocation[0]
        p2738717112: GVL.pieces[0,0].translatedLocation[1]
        OnMouseClick: execute {
            IF(NOT GVL.pieces[0,0].isSelected) THEN
            	// deselect everything
            	FOR i := 0 TO 11 DO
            		GVL.pieces[0,i].isSelected := FALSE;
            		GVL.pieces[1,i].isSelected := FALSE;
            	END_FOR
            	// select the piece
            	GVL.pieces[0,0].isSelected := TRUE;
            	GVL.selectedPieceValidMoveArr := GVL.pieces[0,0].validMoveArr;
            ELSE
            	GVL.pieces[0,0].isSelected := FALSE;
            	GVL.selectedPieceValidMoveArr := GVL.noValidMoveArr;
            END_IF
        }
    Ellipse (440,10 50x50), "%s", text variable: GVL.pieces[1,11].kingText, colour toggle: GVL.pieces[1,11].isSelected
        p3560616238: GVL.pieces[1,11].translatedLocation[0]
        p2738717112: GVL.pieces[1,11].translatedLocation[1]
        OnMouseClick: execute {
            IF(NOT GVL.pieces[1,11].isSelected) THEN
            	// deselect everything
            	FOR i := 0 TO 11 DO
            		GVL.pieces[0,i].isSelected := FALSE;
            		GVL.pieces[1,i].isSelected := FALSE;
            	END_FOR
            	// select the piece
            	GVL.pieces[1,11].isSelected := TRUE;
            	GVL.selectedPieceValidMoveArr := GVL.pieces[1,11].validMoveArr;
            ELSE
            	GVL.pieces[1,11].isSelected := FALSE;
            	GVL.selectedPieceValidMoveArr := GVL.noValidMoveArr;
            END_IF
        }
    Ellipse (440,10 50x50), "%s", text variable: GVL.pieces[1,10].kingText, colour toggle: GVL.pieces[1,10].isSelected
        p3560616238: GVL.pieces[1,10].translatedLocation[0]
        p2738717112: GVL.pieces[1,10].translatedLocation[1]
        OnMouseClick: execute {
            IF(NOT GVL.pieces[1,10].isSelected) THEN
            	// deselect everything
            	FOR i := 0 TO 11 DO
            		GVL.pieces[0,i].isSelected := FALSE;
            		GVL.pieces[1,i].isSelected := FALSE;
            	END_FOR
            	// select the piece
            	GVL.pieces[1,10].isSelected := TRUE;
            	GVL.selectedPieceValidMoveArr := GVL.pieces[1,10].validMoveArr;
            ELSE
            	GVL.pieces[1,10].isSelected := FALSE;
            	GVL.selectedPieceValidMoveArr := GVL.noValidMoveArr;
            END_IF
        }
    Ellipse (540,10 50x50), "%s", text variable: GVL.pieces[1,9].kingText, colour toggle: GVL.pieces[1,9].isSelected
        p3560616238: GVL.pieces[1,9].translatedLocation[0]
        p2738717112: GVL.pieces[1,9].translatedLocation[1]
        OnMouseClick: execute {
            IF(NOT GVL.pieces[1,9].isSelected) THEN
            	// deselect everything
            	FOR i := 0 TO 11 DO
            		GVL.pieces[0,i].isSelected := FALSE;
            		GVL.pieces[1,i].isSelected := FALSE;
            	END_FOR
            	// select the piece
            	GVL.pieces[1,9].isSelected := TRUE;
            	GVL.selectedPieceValidMoveArr := GVL.pieces[1,9].validMoveArr;
            ELSE
            	GVL.pieces[1,9].isSelected := FALSE;
            	GVL.selectedPieceValidMoveArr := GVL.noValidMoveArr;
            END_IF
        }
    Ellipse (540,10 50x50), "%s", text variable: GVL.pieces[1,8].kingText, colour toggle: GVL.pieces[1,8].isSelected
        p3560616238: GVL.pieces[1,8].translatedLocation[0]
        p2738717112: GVL.pieces[1,8].translatedLocation[1]
        OnMouseClick: execute {
            IF(NOT GVL.pieces[1,8].isSelected) THEN
            	// deselect everything
            	FOR i := 0 TO 11 DO
            		GVL.pieces[0,i].isSelected := FALSE;
            		GVL.pieces[1,i].isSelected := FALSE;
            	END_FOR
            	// select the piece
            	GVL.pieces[1,8].isSelected := TRUE;
            	GVL.selectedPieceValidMoveArr := GVL.pieces[1,8].validMoveArr;
            ELSE
            	GVL.pieces[1,8].isSelected := FALSE;
            	GVL.selectedPieceValidMoveArr := GVL.noValidMoveArr;
            END_IF
        }
    Ellipse (540,10 50x50), "%s", text variable: GVL.pieces[1,7].kingText, colour toggle: GVL.pieces[1,7].isSelected
        p3560616238: GVL.pieces[1,7].translatedLocation[0]
        p2738717112: GVL.pieces[1,7].translatedLocation[1]
        OnMouseClick: execute {
            IF(NOT GVL.pieces[1,7].isSelected) THEN
            	// deselect everything
            	FOR i := 0 TO 11 DO
            		GVL.pieces[0,i].isSelected := FALSE;
            		GVL.pieces[1,i].isSelected := FALSE;
            	END_FOR
            	// select the piece
            	GVL.pieces[1,7].isSelected := TRUE;
            	GVL.selectedPieceValidMoveArr := GVL.pieces[1,7].validMoveArr;
            ELSE
            	GVL.pieces[1,7].isSelected := FALSE;
            	GVL.selectedPieceValidMoveArr := GVL.noValidMoveArr;
            END_IF
        }
    Ellipse (540,10 50x50), "%s", text variable: GVL.pieces[1,6].kingText, colour toggle: GVL.pieces[1,6].isSelected
        p3560616238: GVL.pieces[1,6].translatedLocation[0]
        p2738717112: GVL.pieces[1,6].translatedLocation[1]
        OnMouseClick: execute {
            IF(NOT GVL.pieces[1,6].isSelected) THEN
            	// deselect everything
            	FOR i := 0 TO 11 DO
            		GVL.pieces[0,i].isSelected := FALSE;
            		GVL.pieces[1,i].isSelected := FALSE;
            	END_FOR
            	// select the piece
            	GVL.pieces[1,6].isSelected := TRUE;
            	GVL.selectedPieceValidMoveArr := GVL.pieces[1,6].validMoveArr;
            ELSE
            	GVL.pieces[1,6].isSelected := FALSE;
            	GVL.selectedPieceValidMoveArr := GVL.noValidMoveArr;
            END_IF
        }
    Ellipse (540,10 50x50), "%s", text variable: GVL.pieces[1,5].kingText, colour toggle: GVL.pieces[1,5].isSelected
        p3560616238: GVL.pieces[1,5].translatedLocation[0]
        p2738717112: GVL.pieces[1,5].translatedLocation[1]
        OnMouseClick: execute {
            IF(NOT GVL.pieces[1,5].isSelected) THEN
            	// deselect everything
            	FOR i := 0 TO 11 DO
            		GVL.pieces[0,i].isSelected := FALSE;
            		GVL.pieces[1,i].isSelected := FALSE;
            	END_FOR
            	// select the piece
            	GVL.pieces[1,5].isSelected := TRUE;
            	GVL.selectedPieceValidMoveArr := GVL.pieces[1,5].validMoveArr;
            ELSE
            	GVL.pieces[1,5].isSelected := FALSE;
            	GVL.selectedPieceValidMoveArr := GVL.noValidMoveArr;
            END_IF
        }
    Ellipse (640,10 50x50), "%s", text variable: GVL.pieces[1,4].kingText, colour toggle: GVL.pieces[1,4].isSelected
        p3560616238: GVL.pieces[1,4].translatedLocation[0]
        p2738717112: GVL.pieces[1,4].translatedLocation[1]
        OnMouseClick: execute {
            IF(NOT GVL.pieces[1,4].isSelected) THEN
            	// deselect everything
            	FOR i := 0 TO 11 DO
            		GVL.pieces[0,i].isSelected := FALSE;
            		GVL.pieces[1,i].isSelected := FALSE;
            	END_FOR
            	// select the piece
            	GVL.pieces[1,4].isSelected := TRUE;
            	GVL.selectedPieceValidMoveArr := GVL.pieces[1,4].validMoveArr;
            ELSE
            	GVL.pieces[1,4].isSelected := FALSE;
            	GVL.selectedPieceValidMoveArr := GVL.noValidMoveArr;
            END_IF
        }
    Ellipse (640,10 50x50), "%s", text variable: GVL.pieces[1,3].kingText, colour toggle: GVL.pieces[1,3].isSelected
        p3560616238: GVL.pieces[1,3].translatedLocation[0]
        p2738717112: GVL.pieces[1,3].translatedLocation[1]
        OnMouseClick: execute {
            IF(NOT GVL.pieces[1,3].isSelected) THEN
            	// deselect everything
            	FOR i := 0 TO 11 DO
            		GVL.pieces[0,i].isSelected := FALSE;
            		GVL.pieces[1,i].isSelected := FALSE;
            	END_FOR
            	// select the piece
            	GVL.pieces[1,3].isSelected := TRUE;
            	GVL.selectedPieceValidMoveArr := GVL.pieces[1,3].validMoveArr;
            ELSE
            	GVL.pieces[1,3].isSelected := FALSE;
            	GVL.selectedPieceValidMoveArr := GVL.noValidMoveArr;
            END_IF
        }
    Ellipse (640,10 50x50), "%s", text variable: GVL.pieces[1,2].kingText, colour toggle: GVL.pieces[1,2].isSelected
        p3560616238: GVL.pieces[1,2].translatedLocation[0]
        p2738717112: GVL.pieces[1,2].translatedLocation[1]
        OnMouseClick: execute {
            IF(NOT GVL.pieces[1,2].isSelected) THEN
            	// deselect everything
            	FOR i := 0 TO 11 DO
            		GVL.pieces[0,i].isSelected := FALSE;
            		GVL.pieces[1,i].isSelected := FALSE;
            	END_FOR
            	// select the piece
            	GVL.pieces[1,2].isSelected := TRUE;
            	GVL.selectedPieceValidMoveArr := GVL.pieces[1,2].validMoveArr;
            ELSE
            	GVL.pieces[1,2].isSelected := FALSE;
            	GVL.selectedPieceValidMoveArr := GVL.noValidMoveArr;
            END_IF
        }
    Ellipse (640,10 50x50), "%s", text variable: GVL.pieces[1,1].kingText, colour toggle: GVL.pieces[1,1].isSelected
        p3560616238: GVL.pieces[1,1].translatedLocation[0]
        p2738717112: GVL.pieces[1,1].translatedLocation[1]
        OnMouseClick: execute {
            IF(NOT GVL.pieces[1,1].isSelected) THEN
            	// deselect everything
            	FOR i := 0 TO 11 DO
            		GVL.pieces[0,i].isSelected := FALSE;
            		GVL.pieces[1,i].isSelected := FALSE;
            	END_FOR
            	// select the piece
            	GVL.pieces[1,1].isSelected := TRUE;
            	GVL.selectedPieceValidMoveArr := GVL.pieces[1,1].validMoveArr;
            ELSE
            	GVL.pieces[1,1].isSelected := FALSE;
            	GVL.selectedPieceValidMoveArr := GVL.noValidMoveArr;
            END_IF
        }
    Ellipse (640,10 50x50), "%s", text variable: GVL.pieces[1,9].kingText, colour toggle: GVL.pieces[1,0].isSelected
        p3560616238: GVL.pieces[1,0].translatedLocation[0]
        p2738717112: GVL.pieces[1,0].translatedLocation[1]
        OnMouseClick: execute {
            IF(NOT GVL.pieces[1,0].isSelected) THEN
            	// deselect everything
            	FOR i := 0 TO 11 DO
            		GVL.pieces[0,i].isSelected := FALSE;
            		GVL.pieces[1,i].isSelected := FALSE;
            	END_FOR
            	// select the piece
            	GVL.pieces[1,0].isSelected := TRUE;
            	GVL.selectedPieceValidMoveArr := GVL.pieces[1,0].validMoveArr;
            ELSE
            	GVL.pieces[1,0].isSelected := FALSE;
            	GVL.selectedPieceValidMoveArr := GVL.noValidMoveArr;
            END_IF
        }
    Button (774,116 150x30), "Setup Board"
        tap Gameplay.commenceSetup
    Button (778,184 150x30), "Switch Turns"
        OnMouseClick:  ToggleVariable=GVL.redsTurn
    Textfield (780,250 150x30), "%d", text variable: GVL.blackPiecesTaken
END_VISUALIZATION
